                      if linea == 1:
                          P_Tipo1[NMovAct[linea-1]-1] = P_Tipo1[ordenM9_T1[NMovAct[linea-1]-1]-1]
                          P_Tipo2[NMovAct[linea-1]-1] = P_Tipo2[ordenM9_T2[NMovAct[linea-1]-1]-1]
                      end
                    else:
                      $ 709 "ElseIf Rec_Mosaico[Programa_1-1]≟10"
                      if (Rec_Mosaico[Programa_1-1] == 10):
                        $ 710 "Mosaico 10"
                        $ 716 "Script: mosaico10.script"
                        #MOSAICO 10
                        #P_Tipo1 y P_Tipo2 tienen que venir ya relativizados del asistente!

                        if ModificarMos == True:

                        	P_Tipo1_Mos10 = P_Tipo1
                        	P_Tipo2_Mos10 = P_Tipo2
                        	ordenM10_T1 = orden_T1
                        	ordenM10_T2 = orden_T2

                        end

                        ModificarMos = False

                        P_Tipo1 = P_Tipo1_Mos10
                        P_Tipo2 = P_Tipo2_Mos10


                        #En caso de que actualice movimientos de 2 en 2 (modificación de mosaico o crear nuevo)
                        if Cogida2en2 == True:

                        	Movs2en2_M10_T1 = Movs2en2_Tipo1
                        	Movs2en2_M10_T2 = Movs2en2_Tipo2

                        end

                        Cogida2en2 = False

                        #Siempre, si hay algún movimiento doble, actualizo si el movimiento actual lo es o no
                        if Rec_Cogida2en2[Programa-1] == True:
                        	if Rec_TipoCapa[NCapaAct[linea-1]-1] == 1:
                        		Movs2en2 = Movs2en2_M10_T1
                        		if linea == 1:
                        			Movs2en2[NMovAct[linea-1]-1] = Movs2en2[ordenM10_T1[NMovAct[linea-1]-1]-1]
                        		end
                        	else:
                        		Movs2en2 = Movs2en2_M10_T2
                        		if linea == 1:
                        			Movs2en2[NMovAct[linea-1]-1] = Movs2en2[ordenM10_T2[NMovAct[linea-1]-1]-1]
                        		end
                        	end
                        else:
                        	Movs2en2[NMovAct[linea-1]-1] = False
                        end

                        if linea == 1:
                            P_Tipo1[NMovAct[linea-1]-1] = P_Tipo1[ordenM10_T1[NMovAct[linea-1]-1]-1]
                            P_Tipo2[NMovAct[linea-1]-1] = P_Tipo2[ordenM10_T2[NMovAct[linea-1]-1]-1]
                        end
                      else:
                        $ 717 "ElseIf Rec_Mosaico[Programa_1-1]≟11"
                        if (Rec_Mosaico[Programa_1-1] == 11):
                          $ 718 "Mosaico 11"
                          $ 724 "Script: mosaico11.script"
                          #MOSAICO 10
                          #P_Tipo1 y P_Tipo2 tienen que venir ya relativizados del asistente!

                          if ModificarMos == True:

                          	P_Tipo1_Mos11 = P_Tipo1
                          	P_Tipo2_Mos11 = P_Tipo2
                          	ordenM11_T1 = orden_T1
                          	ordenM11_T2 = orden_T2

                          end

                          ModificarMos = False

                          P_Tipo1 = P_Tipo1_Mos11
                          P_Tipo2 = P_Tipo2_Mos11


                          #En caso de que actualice movimientos de 2 en 2 (modificación de mosaico o crear nuevo)
                          if Cogida2en2 == True:

                          	Movs2en2_M11_T1 = Movs2en2_Tipo1
                          	Movs2en2_M11_T2 = Movs2en2_Tipo2

                          end

                          Cogida2en2 = False

                          #Siempre, si hay algún movimiento doble, actualizo si el movimiento actual lo es o no
                          if Rec_Cogida2en2[Programa_1-1] == True:
                          	if Rec_TipoCapa[NCapaAct[linea-1]-1] == 1:
                          		Movs2en2 = Movs2en2_M11_T1
                          		if linea == 1:
                          			Movs2en2[NMovAct[linea-1]-1] = Movs2en2[ordenM11_T1[NMovAct[linea-1]-1]-1]
                          		end
                          	else:
                          		Movs2en2 = Movs2en2_M11_T2
                          		if linea == 1:
                          			Movs2en2[NMovAct[linea-1]-1] = Movs2en2[ordenM11_T2[NMovAct[linea-1]-1]-1]
                          		end
                          	end
                          else:
                          	Movs2en2[NMovAct[linea-1]-1] = False
                          end

                          if linea == 1:
                              P_Tipo1[NMovAct[linea-1]-1] = P_Tipo1[ordenM11_T1[NMovAct[linea-1]-1]-1]
                              P_Tipo2[NMovAct[linea-1]-1] = P_Tipo2[ordenM11_T2[NMovAct[linea-1]-1]-1]
                          end
                        else:
                          $ 725 "ElseIf Rec_Mosaico[Programa_1-1]≟12"
                          if (Rec_Mosaico[Programa_1-1] == 12):
                            $ 726 "Mosaico 12"
                            $ 796 "Script: mosaico12.script"
                            #MOSAICO 10
                            #P_Tipo1 y P_Tipo2 tienen que venir ya relativizados del asistente!

                            if ModificarMos == True:

                            	P_Tipo1_Mos12 = P_Tipo1
                            	P_Tipo2_Mos12 = P_Tipo2
                            	ordenM12_T1 = orden_T1
                            	ordenM12_T2 = orden_T2

                            end

                            ModificarMos = False

                            P_Tipo1 = P_Tipo1_Mos12
                            P_Tipo2 = P_Tipo2_Mos12


                            #En caso de que actualice movimientos de 2 en 2 (modificación de mosaico o crear nuevo)
                            if Cogida2en2 == True:

                            	Movs2en2_M12_T1 = Movs2en2_Tipo1
                            	Movs2en2_M12_T2 = Movs2en2_Tipo2

                            end

                            Cogida2en2 = False

                            #Siempre, si hay algún movimiento doble, actualizo si el movimiento actual lo es o no
                            if Rec_Cogida2en2[Programa_1-1] == True:
                            	if Rec_TipoCapa[NCapaAct[linea-1]-1] == 1:
                            		Movs2en2 = Movs2en2_M12_T1
                            		if linea == 1:
                            			Movs2en2[NMovAct[linea-1]-1] = Movs2en2[ordenM12_T1[NMovAct[linea-1]-1]-1]
                            		end
                            	else:
                            		Movs2en2 = Movs2en2_M12_T2
                            		if linea == 1:
                            			Movs2en2[NMovAct[linea-1]-1] = Movs2en2[ordenM12_T2[NMovAct[linea-1]-1]-1]
                            		end
                            	end
                            else:
                            	Movs2en2[NMovAct[linea-1]-1] = False
                            end

                            if linea == 1:
                                P_Tipo1[NMovAct[linea-1]-1] = P_Tipo1[ordenM12_T1[NMovAct[linea-1]-1]-1]
                                P_Tipo2[NMovAct[linea-1]-1] = P_Tipo2[ordenM12_T2[NMovAct[linea-1]-1]-1]
                            end
                          else:
                            $ 797 "Else" "noBreak"
                            $ 798 "Popup: Número de mosaico elegido no válido. Contacta con Geniotic."
                            popup("Número de mosaico elegido no válido. Contacta con Geniotic.", "Mensaje", False, False, blocking=True)
                            $ 799 "Halt"
                            halt
                          end
                        end
                      end
                    end
                  end
                end
              end
            end
          end
        end
      end
    end
  end
  def Cambios():
    $ 800 "Cambios" "noBreak"
    $ 801 "StepCode = 5"
    StepCode = 5
    $ 802 "If CambioPrograma"
    if (CambioPrograma):
      $ 803 "write_output_boolean_register(5,False)"
      write_output_boolean_register(5,False)
      $ 804 "'CambiosPrograma = False'"
      # 'CambiosPrograma = False'
      $ 809 "PonerCarton = [False,False]"
      PonerCarton = [False,False]
      $ 810 "Confirmacion = request_boolean_from_primary_client(' Al cambiar de programa se inicializan los contadores, ¿quieres continuar? ')"
      Confirmacion = request_boolean_from_primary_client(" Al cambiar de programa se inicializan los contadores, ¿quieres continuar? ")
      $ 811 "If Confirmacion"
      if (Confirmacion):
        $ 812 "Confirmacion = False"
        Confirmacion = False
        $ 813 "If (NCapaAct[0] ≠1 or NMovAct[0]≠1)"
        if ((NCapaAct[0]  != 1  or  NMovAct[0] != 1)):
          $ 814 "palet_completo(0)"
          palet_completo(0)
        end
        $ 815 "If (NCapaAct[1] ≠1 or NMovAct[1]≠1)"
        if ((NCapaAct[1]  != 1  or  NMovAct[1] != 1)):
          $ 816 "palet_completo(1)"
          palet_completo(1)
        end
        $ 817 "Wait: 0.01"
        sleep(0.01)
        $ 818 "aux = request_integer_from_primary_client('Elige programa [1-12]')"
        aux = request_integer_from_primary_client("Elige programa [1-12]")
        $ 819 "Wait: 0.01"
        sleep(0.01)
        $ 820 "Loop aux<1 or aux>12"
        while (aux<1 or aux>12):
          $ 821 "aux = request_integer_from_primary_client('Elige programa válido [1-12]')"
          aux = request_integer_from_primary_client("Elige programa válido [1-12]")
          $ 822 "sync()"
          sync()
        end
        $ 823 "If Rec_Mosaico[aux-1]≟0"
        if (Rec_Mosaico[aux-1] == 0):
          $ 824 "popup(' Programa vacío. Creálo o cambia a otro programa', title = ' Programa vacío', blocking = True)"
          popup(" Programa vacío. Creálo o cambia a otro programa", title = " Programa vacío", blocking = True)
        else:
          $ 825 "Else" "noBreak"
          $ 826 "Programa_1 = aux"
          Programa_1 = aux
        end
        $ 827 "NPaletAct = 0"
        NPaletAct = 0
        $ 828 "pop_up('¡Cambios finalizados!',3,False)"
        pop_up("¡Cambios finalizados!",3,False)
      end
    end
    $ 829 "If CambiosAvanzados"
    if (CambiosAvanzados):
      $ 830 "write_output_boolean_register(6,False)"
      write_output_boolean_register(6,False)
      $ 831 "'CambiosAvanzados = False'"
      # 'CambiosAvanzados = False'
      $ 832 "movej(Home_q,0.5,0.5,0,0)"
      movej(Home_q,0.5,0.5,0,0)
      $ 836 "aux = request_integer_from_primary_client(' Introduce la contraseña ')"
      aux = request_integer_from_primary_client(" Introduce la contraseña ")
      $ 837 "If aux≟1234"
      if (aux == 1234):
        $ 838 "Cambio_2≔0"
        global Cambio_2=0
        $ 839 "Loop Cambio_2≟0"
        while (Cambio_2 == 0):
          $ 840 "Cambio = request_integer_from_primary_client('Modificar programa [1], cambiar contadores [2] o ajustar un mov [3]?')"
          Cambio = request_integer_from_primary_client("Modificar programa [1], cambiar contadores [2] o ajustar un mov [3]?")
          $ 841 "Wait: 0.5"
          sleep(0.5)
          $ 842 "Loop Cambio<1 or Cambio>3"
          while (Cambio<1  or  Cambio>3):
            $ 843 "Cambio = request_integer_from_primary_client('Modificar programa [1], cambiar contadores [2] o ajustar un mov [3]?')"
            Cambio = request_integer_from_primary_client("Modificar programa [1], cambiar contadores [2] o ajustar un mov [3]?")
            $ 844 "sync()"
            sync()
          end
          $ 845 "If Cambio≟1"
          if (Cambio == 1):
            $ 846 "StepCode = 6"
            StepCode = 6
            $ 847 "Modificar_Programa"
            $ 848 "Confirmacion = request_boolean_from_primary_client(' Al cambiar de programa se inicializan los contadores, ¿quieres continuar? ')"
            Confirmacion = request_boolean_from_primary_client(" Al cambiar de programa se inicializan los contadores, ¿quieres continuar? ")
            $ 849 "If Confirmacion"
            if (Confirmacion):
              $ 850 "Confirmacion = False"
              Confirmacion = False
              $ 851 "If (NCapaAct[0] ≠1 or NMovAct[0]≠1)"
              if ((NCapaAct[0]  != 1  or  NMovAct[0] != 1)):
                $ 852 "palet_completo(0)"
                palet_completo(0)
              end
              $ 853 "If (NCapaAct[1] ≠1 or NMovAct[1]≠1)"
              if ((NCapaAct[1]  != 1  or  NMovAct[1] != 1)):
                $ 854 "palet_completo(1)"
                palet_completo(1)
              end
              $ 855 "Wait: 0.01"
              sleep(0.01)
              $ 856 "aux = request_integer_from_primary_client('Elige programa [1-12]')"
              aux = request_integer_from_primary_client("Elige programa [1-12]")
              $ 857 "Wait: 0.01"
              sleep(0.01)
              $ 858 "Loop aux<1 or aux>12"
              while (aux<1 or aux>12):
                $ 859 "aux = request_integer_from_primary_client('Elige programa válido [1-12]')"
                aux = request_integer_from_primary_client("Elige programa válido [1-12]")
                $ 860 "sync()"
                sync()
              end
              $ 861 "Loop Rec_Mosaico[aux-1]≟0 and ProgNuevo≟ False "
              while (Rec_Mosaico[aux-1] == 0  and  ProgNuevo ==   False  ):
                $ 862 "ProgNuevo = request_boolean_from_primary_client('Programa vacío. ¿Quieres crear uno nuevo [Sí] o elegir otro programa a modificar [No]?')"
                ProgNuevo = request_boolean_from_primary_client("Programa vacío. ¿Quieres crear uno nuevo [Sí] o elegir otro programa a modificar [No]?")
                $ 863 "If ProgNuevo≟ False "
                if (ProgNuevo ==   False  ):
                  $ 864 "aux = request_integer_from_primary_client('Elige programa [1-12]')"
                  aux = request_integer_from_primary_client("Elige programa [1-12]")
                  $ 865 "Loop aux<1 or aux>12"
                  while (aux<1 or aux>12):
                    $ 866 "aux = request_integer_from_primary_client('Elige programa válido [1-12]')"
                    aux = request_integer_from_primary_client("Elige programa válido [1-12]")
                    $ 867 "sync()"
                    sync()
                  end
                end
                $ 868 "sync()"
                sync()
              end
              $ 869 "ProgNuevo = False"
              ProgNuevo = False
              $ 870 "NPaletAct = 0"
              NPaletAct = 0
              $ 871 "Programa_1 = aux"
              Programa_1 = aux
              $ 872 "Modificaciones"
              $ 873 "aux_bool = request_boolean_from_primary_client(' ¿Quieres modificar el punto de cogida?')"
              aux_bool = request_boolean_from_primary_client(" ¿Quieres modificar el punto de cogida?")
              $ 874 "If aux_bool"
              if (aux_bool):
                $ 875 "freedrive_mode()"
                freedrive_mode()
                $ 876 "popup('Ve al punto y presiona Continuar', 'Punto cogida', False, False, blocking=True)"
                popup("Ve al punto y presiona Continuar", "Punto cogida", False, False, blocking=True)
                $ 877 "end_freedrive_mode()"
                end_freedrive_mode()
                $ 878 "PuntosCogida[Programa_1-1]=get_actual_tcp_pose()"
                PuntosCogida[Programa_1-1]= get_actual_tcp_pose ()
                $ 879 "popup('Mueve el robot a un sitio seguro antes de ir a Home', 'Mensaje', False, False, blocking=True)"
                popup("Mueve el robot a un sitio seguro antes de ir a Home", "Mensaje", False, False, blocking=True)
                $ 880 "movej(Home_q,0.5,0.5,0,0)"
                movej(Home_q,0.5,0.5,0,0)
              end
              $ 881 "aux=request_integer_from_primary_client('Largo producto (mm)')"
              aux=request_integer_from_primary_client("Largo producto (mm)")
              $ 882 "Rec_LargoPrd[Programa_1-1]=aux"
              Rec_LargoPrd[Programa_1-1]=aux
              $ 883 "Wait: 0.5"
              sleep(0.5)
              $ 884 "aux=request_integer_from_primary_client('Ancho producto (mm)')"
              aux=request_integer_from_primary_client("Ancho producto (mm)")
              $ 885 "Rec_AnchoPrd[Programa_1-1]=aux"
              Rec_AnchoPrd[Programa_1-1]=aux
              $ 886 "Wait: 0.5"
              sleep(0.5)
              $ 887 "aux_float=request_float_from_primary_client('Alto producto (mm)')"
              aux_float=request_float_from_primary_client("Alto producto (mm)")
              $ 888 "Rec_AltoPrd[Programa_1-1]=aux_float"
              Rec_AltoPrd[Programa_1-1]=aux_float
              $ 889 "Wait: 0.5"
              sleep(0.5)
              $ 890 "aux=request_integer_from_primary_client('Número de movimientos por capa')"
              aux=request_integer_from_primary_client("Número de movimientos por capa")
              $ 891 "Rec_NMovsCapa[Programa_1-1]=aux"
              Rec_NMovsCapa[Programa_1-1]=aux
              $ 892 "Wait: 0.5"
              sleep(0.5)
              $ 893 "aux=request_integer_from_primary_client('Número de capas totales')"
              aux=request_integer_from_primary_client("Número de capas totales")
              $ 894 "Rec_NCapasTot[Programa_1-1]=aux"
              Rec_NCapasTot[Programa_1-1]=aux
              $ 895 "Wait: 0.5"
              sleep(0.5)
              $ 896 "aux_bool=request_boolean_from_primary_client('¿Capas trabadas?')"
              aux_bool=request_boolean_from_primary_client("¿Capas trabadas?")
              $ 897 "Rec_CapasTrab[Programa_1-1]=aux_bool"
              Rec_CapasTrab[Programa_1-1]=aux_bool
              $ 898 "Wait: 0.5"
              sleep(0.5)
              $ 899 "aux_float=request_float_from_primary_client('Peso producto (kg)')"
              aux_float=request_float_from_primary_client("Peso producto (kg)")
              $ 900 "Rec_PesoPrd[Programa_1-1]=aux_float"
              Rec_PesoPrd[Programa_1-1]=aux_float
              $ 901 "Wait: 0.5"
              sleep(0.5)
              $ 902 "aux_bool=request_boolean_from_primary_client('¿Quieres usar un mosaico existente [Sí] o modificar/crear un mosaico [No]?')"
              aux_bool=request_boolean_from_primary_client("¿Quieres usar un mosaico existente [Sí] o modificar/crear un mosaico [No]?")
              $ 903 "ModificarMos = not(aux_bool)"
              ModificarMos = not(aux_bool)
              $ 904 "Wait: 0.5"
              sleep(0.5)
              $ 905 "aux=request_integer_from_primary_client('Elige un mosaico [1-12]')"
              aux=request_integer_from_primary_client("Elige un mosaico [1-12]")
              $ 906 "Loop aux<1 or aux>12"
              while (aux<1  or  aux>12):
                $ 907 "aux=request_integer_from_primary_client('Elige un mosaico válido [1-12]')"
                aux=request_integer_from_primary_client("Elige un mosaico válido [1-12]")
                $ 908 "sync()"
                sync()
              end
              $ 909 "Wait: 0.5"
              sleep(0.5)
              $ 910 "Rec_Mosaico[Programa_1-1]=aux"
              Rec_Mosaico[Programa_1-1]=aux
              $ 911 "Modificar mosaico"
              $ 912 "If ModificarMos"
              if (ModificarMos):
                $ 913 "i≔0"
                global i=0
                $ 914 "popup('Presiona Continuar para grabar los movimientos de la primera capa', 'Ajuste mosaico tipo capa 1', False, False, blocking=True)"
                popup("Presiona Continuar para grabar los movimientos de la primera capa", "Ajuste mosaico tipo capa 1", False, False, blocking=True)
                $ 915 "Loop i<Rec_NMovsCapa[Programa_1-1]"
                while (i<Rec_NMovsCapa[Programa_1-1]):
                  $ 916 "freedrive_mode()"
                  freedrive_mode()
                  $ 917 "popup('Mueve el robot al movimiento ' + to_str(i+1) + ' y presiona Continuar', title = ' Ajuste mosaico tipo capa 1', blocking = True)"
                  popup("Mueve el robot al movimiento " + to_str(i+1) + " y presiona Continuar", title = " Ajuste mosaico tipo capa 1", blocking = True)
                  $ 918 "end_freedrive_mode()"
                  end_freedrive_mode()
                  $ 919 "P_Tipo1[i] = get_actual_tcp_pose()"
                  P_Tipo1[i] =  get_actual_tcp_pose ()
                  $ 920 "i = i + 1"
                  i = i + 1
                  $ 921 "sync()"
                  sync()
                end
                $ 922 "i=0"
                i=0
                $ 923 "If Rec_CapasTrab[Programa_1-1]"
                if (Rec_CapasTrab[Programa_1-1]):
                  $ 924 "popup('Presiona Continuar para grabar los movimientos de la segunda capa', 'Ajuste mosaico tipo capa 2', False, False, blocking=True)"
                  popup("Presiona Continuar para grabar los movimientos de la segunda capa", "Ajuste mosaico tipo capa 2", False, False, blocking=True)
                  $ 925 "Loop i<Rec_NMovsCapa[Programa_1-1]"
                  while (i<Rec_NMovsCapa[Programa_1-1]):
                    $ 926 "freedrive_mode()"
                    freedrive_mode()
                    $ 927 "popup('Mueve el robot al movimiento ' + to_str(i+1) + ' y presiona Continuar', title = ' Ajuste mosaico tipo capa 2', blocking = True)"
                    popup("Mueve el robot al movimiento " + to_str(i+1) + " y presiona Continuar", title = " Ajuste mosaico tipo capa 2", blocking = True)
                    $ 928 "end_freedrive_mode()"
                    end_freedrive_mode()
                    $ 929 "P_Tipo2[i] = get_actual_tcp_pose()"
                    P_Tipo2[i] =  get_actual_tcp_pose ()
                    $ 930 "i = i + 1"
                    i = i + 1
                    $ 931 "sync()"
                    sync()
                  end
                end
                $ 932 "freedrive_mode()"
                freedrive_mode()
                $ 933 "popup('Mueve el robot a un sitio seguro antes de ir a Home', 'Mensaje', False, False, blocking=True)"
                popup("Mueve el robot a un sitio seguro antes de ir a Home", "Mensaje", False, False, blocking=True)
                $ 934 "end_freedrive_mode()"
                end_freedrive_mode()
                $ 935 "Wait: 0.5"
                sleep(0.5)
                $ 936 "Script: Relativizar.script"
                #Tras grabar los puntos
                local k = 0
                while k < 25:
                    P_Tipo1[k] = pose_trans(Pbf,P_Tipo1[k])
                    P_Tipo2[k] = pose_trans(Pbf,P_Tipo2[k])
                    k = k + 1
                end
                $ 937 "movej(Home_q,0.5,0.5,0,0)"
                movej(Home_q,0.5,0.5,0,0)
                $ 938 "Orden"
                $ 939 "aux = 0"
                aux = 0
                $ 940 "popup('Al presionar Continuar vamos a configurar los mosaicos de la línea 1', 'Mensaje', False, False, blocking=True)"
                popup("Al presionar Continuar vamos a configurar los mosaicos de la línea 1", "Mensaje", False, False, blocking=True)
                $ 941 "popup('Presiona Continuar para indicar el orden de los movimientos de la primera capa', 'Mensaje', False, False, blocking=True)"
                popup("Presiona Continuar para indicar el orden de los movimientos de la primera capa", "Mensaje", False, False, blocking=True)
                $ 942 "Loop aux<Rec_NMovsCapa[Programa_1-1]"
                while (aux<Rec_NMovsCapa[Programa_1-1]):
                  $ 943 "orden_T1[aux] = request_integer_from_primary_client(' El movimiento número ' + to_str(aux+1) + ' de la línea 1, ¿con qué número de movimiento se corresponde de la línea 2?')"
                  orden_T1[aux] = request_integer_from_primary_client(" El movimiento número " + to_str(aux+1) + " de la línea 1, ¿con qué número de movimiento se corresponde de la línea 2?")
                  $ 944 "aux = aux +1"
                  aux = aux +1
                  $ 945 "sync()"
                  sync()
                end
                $ 946 "If Rec_CapasTrab[Programa_1-1]"
                if (Rec_CapasTrab[Programa_1-1]):
                  $ 947 "popup('Presiona Continuar para indicar el orden de los movimientos de la segunda capa', 'Mensaje', False, False, blocking=True)"
                  popup("Presiona Continuar para indicar el orden de los movimientos de la segunda capa", "Mensaje", False, False, blocking=True)
                  $ 948 "aux = 0"
                  aux = 0
                  $ 949 "Loop aux<Rec_NMovsCapa[Programa_1-1]"
                  while (aux<Rec_NMovsCapa[Programa_1-1]):
                    $ 950 "orden_T2[aux] = request_integer_from_primary_client(' El movimiento número ' + to_str(aux+1) + ' de la línea 1, ¿con qué número de movimiento se corresponde de la línea 2?')"
                    orden_T2[aux] = request_integer_from_primary_client(" El movimiento número " + to_str(aux+1) + " de la línea 1, ¿con qué número de movimiento se corresponde de la línea 2?")
                    $ 951 "aux = aux +1"
                    aux = aux +1
                    $ 952 "sync()"
                    sync()
                  end
                end
                $ 953 "Cogida2en2=request_boolean_from_primary_client('¿Hay movimientos dobles?')"
                Cogida2en2=request_boolean_from_primary_client("¿Hay movimientos dobles?")
                $ 954 "Rec_Cogida2en2[Programa_1-1]=Cogida2en2"
                Rec_Cogida2en2[Programa_1-1]=Cogida2en2
                $ 955 "Wait: 0.5"
                sleep(0.5)
                $ 956 "Movimientos de 2 en 2"
                $ 957 "If Cogida2en2"
                if (Cogida2en2):
                  $ 958 "aux=request_integer_from_primary_client('¿Cuántos movimientos son dobles?')"
                  aux=request_integer_from_primary_client("¿Cuántos movimientos son dobles?")
                  $ 959 "Loop aux<1 or aux>Rec_NMovsCapa[Programa_1-1]"
                  while (aux<1  or  aux>Rec_NMovsCapa[Programa_1-1]):
                    $ 960 "aux=request_integer_from_primary_client('¿Cuántos movimientos son dobles?')"
                    aux=request_integer_from_primary_client("¿Cuántos movimientos son dobles?")
                    $ 961 "sync()"
                    sync()
                  end
                  $ 962 "aux_2=0"
                  aux_2=0
                  $ 963 "Loop aux_2<aux"
                  while (aux_2<aux):
                    $ 964 "aux_3=request_integer_from_primary_client('Indicar número del siguiente movimiento doble (primera capa)')"
                    aux_3=request_integer_from_primary_client("Indicar número del siguiente movimiento doble (primera capa)")
                    $ 965 "sync()"
                    sync()
                    $ 966 "Loop aux_3<1 or aux_3>Rec_NMovsCapa[Programa_1-1]"
                    while (aux_3<1  or  aux_3>Rec_NMovsCapa[Programa_1-1]):
                      $ 967 "aux_3=request_integer_from_primary_client('Número de movimiento doble incorrecto. Prueba otra vez:')"
                      aux_3=request_integer_from_primary_client("Número de movimiento doble incorrecto. Prueba otra vez:")
                      $ 968 "sync()"
                      sync()
                    end
                    $ 969 "Movs2en2_Tipo1[aux_3-1]= True "
                    Movs2en2_Tipo1[aux_3-1]=  True
                    $ 970 "aux_2=aux_2+1"
                    aux_2=aux_2+1
                  end
                  $ 971 "If Rec_CapasTrab[Programa_1-1]"
                  if (Rec_CapasTrab[Programa_1-1]):
                    $ 972 "aux_2=0"
                    aux_2=0
                    $ 973 "Loop aux_2<aux"
                    while (aux_2<aux):
                      $ 974 "aux_3=request_integer_from_primary_client('Indicar número del siguiente movimiento doble (segunda capa)')"
                      aux_3=request_integer_from_primary_client("Indicar número del siguiente movimiento doble (segunda capa)")
                      $ 975 "sync()"
                      sync()
                      $ 976 "Loop aux_3<1 or aux_3>Rec_NMovsCapa[Programa_1-1]"
                      while (aux_3<1  or  aux_3>Rec_NMovsCapa[Programa_1-1]):
                        $ 977 "aux_3=request_integer_from_primary_client('Número de movimiento doble incorrecto. Prueba otra vez:')"
                        aux_3=request_integer_from_primary_client("Número de movimiento doble incorrecto. Prueba otra vez:")
                        $ 978 "sync()"
                        sync()
                      end
                      $ 979 "Movs2en2_Tipo2[aux_3-1]= True "
                      Movs2en2_Tipo2[aux_3-1]=  True
                      $ 980 "aux_2=aux_2+1"
                      aux_2=aux_2+1
                    end
                  end
                else:
                  $ 981 "Else" "noBreak"
                  $ 982 "aux_bool=request_boolean_from_primary_client('¿Es necesario activar los 2 circuitos de vacío para coger este producto?')"
                  aux_bool=request_boolean_from_primary_client("¿Es necesario activar los 2 circuitos de vacío para coger este producto?")
                  $ 983 "Rec_2Vacios[Programa_1-1] = aux_bool"
                  Rec_2Vacios[Programa_1-1] = aux_bool
                end
              end
            end
          else:
            $ 984 "ElseIf Cambio≟2"
            if (Cambio == 2):
              $ 985 "StepCode = 7"
              StepCode = 7
              $ 986 "Cambio_Contadores"
              $ 987 "aux = request_integer_from_primary_client('Línea [1 - 2]')"
              aux = request_integer_from_primary_client("Línea [1 - 2]")
              $ 988 "Wait: 0.5"
              sleep(0.5)
              $ 989 "Loop aux<1 or aux>2"
              while (aux<1  or  aux>2):
                $ 990 "aux = request_integer_from_primary_client('Línea [1 - 2]')"
                aux = request_integer_from_primary_client("Línea [1 - 2]")
                $ 991 "sync()"
                sync()
              end
              $ 992 "PonerCarton[aux-1] = False"
              PonerCarton[aux-1] = False
              $ 993 "CartonBase[aux-1] = True"
              CartonBase[aux-1] = True
              $ 994 "aux_2 = request_integer_from_primary_client(' Número de capa [1 - ' + to_str(Rec_NCapasTot[Programa_1-1]) +  ']')"
              aux_2 = request_integer_from_primary_client(" Número de capa [1 - " + to_str(Rec_NCapasTot[Programa_1-1]) +  "]")
              $ 995 "Wait: 0.5"
              sleep(0.5)
              $ 996 "Loop aux_2<1 or aux_2>Rec_NCapasTot[Programa_1-1]"
              while (aux_2<1  or  aux_2>Rec_NCapasTot[Programa_1-1]):
                $ 997 "aux_2 = request_integer_from_primary_client(' Número de capa [1 - ' + to_str(Rec_NCapasTot[Programa_1-1]) +  ']')"
                aux_2 = request_integer_from_primary_client(" Número de capa [1 - " + to_str(Rec_NCapasTot[Programa_1-1]) +  "]")
                $ 998 "sync()"
                sync()
              end
              $ 999 "NCapaAct[aux-1] = aux_2"
              NCapaAct[aux-1] = aux_2
              $ 1000 "aux_2= request_integer_from_primary_client(' Número de movimiento [1 - ' + to_str(Rec_NMovsCapa[Programa_1-1]) +  ']')"
              aux_2= request_integer_from_primary_client(" Número de movimiento [1 - " + to_str(Rec_NMovsCapa[Programa_1-1]) +  "]")
              $ 1001 "Wait: 0.5"
              sleep(0.5)
              $ 1002 "Loop aux_2<1 or aux_2>Rec_NMovsCapa[Programa_1-1]"
              while (aux_2<1  or  aux_2>Rec_NMovsCapa[Programa_1-1]):
                $ 1003 "aux_2= request_integer_from_primary_client(' Número de movimiento [1 - ' + to_str(Rec_NMovsCapa[Programa_1-1]) +  ']')"
                aux_2= request_integer_from_primary_client(" Número de movimiento [1 - " + to_str(Rec_NMovsCapa[Programa_1-1]) +  "]")
                $ 1004 "sync()"
                sync()
              end
              $ 1005 "NMovAct[aux-1] = aux_2"
              NMovAct[aux-1] = aux_2
            else:
              $ 1006 "ElseIf Cambio≟3"
              if (Cambio == 3):
                $ 1007 "StepCode = 8"
                StepCode = 8
                $ 1008 "Ajuste de un movimiento"
                $ 1009 "aux_bool = request_boolean_from_primary_client('¿Quieres ajustar un movimiento de dejada [Sí] o cogida [No]?')"
                aux_bool = request_boolean_from_primary_client("¿Quieres ajustar un movimiento de dejada [Sí] o cogida [No]?")
                $ 1010 "Wait: 0.5"
                sleep(0.5)
                $ 1011 "If aux_bool"
                if (aux_bool):
                  $ 1012 "If Rec_CapasTrab[Programa_1-1]≟ True "
                  if (Rec_CapasTrab[Programa_1-1] ==   True  ):
                    $ 1013 "Ajuste_TipoCapa = request_integer_from_primary_client('Elige el tipo de capa a ajustar [1 - 2]')"
                    Ajuste_TipoCapa = request_integer_from_primary_client("Elige el tipo de capa a ajustar [1 - 2]")
                    $ 1014 "Wait: 0.5"
                    sleep(0.5)
                    $ 1015 "Loop Ajuste_TipoCapa<1 or Ajuste_TipoCapa>2"
                    while (Ajuste_TipoCapa<1  or  Ajuste_TipoCapa>2):
                      $ 1016 "Ajuste_TipoCapa = request_integer_from_primary_client('Elige el tipo de capa a ajustar [1 - 2]')"
                      Ajuste_TipoCapa = request_integer_from_primary_client("Elige el tipo de capa a ajustar [1 - 2]")
                      $ 1017 "sync()"
                      sync()
                    end
                  else:
                    $ 1018 "Else" "noBreak"
                    $ 1019 "Ajuste_TipoCapa = 1"
                    Ajuste_TipoCapa = 1
                  end
                  $ 1020 "Ajuste_NumMov = request_integer_from_primary_client(' ¿Qué movimiento quieres ajustar? [1-' +to_str(Rec_NMovsCapa[Programa_1-1])+']')"
                  Ajuste_NumMov = request_integer_from_primary_client(" ¿Qué movimiento quieres ajustar? [1-" +to_str(Rec_NMovsCapa[Programa_1-1])+"]")
                  $ 1021 "Wait: 0.5"
                  sleep(0.5)
                  $ 1022 "Loop Ajuste_NumMov<1 or Ajuste_NumMov>Rec_NMovsCapa[Programa_1-1]"
                  while (Ajuste_NumMov<1  or  Ajuste_NumMov>Rec_NMovsCapa[Programa_1-1]):
                    $ 1023 "Ajuste_NumMov = request_integer_from_primary_client(' ¿Qué movimiento quieres ajustar? [1-' +to_str(Rec_NMovsCapa[Programa_1-1])+']')"
                    Ajuste_NumMov = request_integer_from_primary_client(" ¿Qué movimiento quieres ajustar? [1-" +to_str(Rec_NMovsCapa[Programa_1-1])+"]")
                    $ 1024 "sync()"
                    sync()
                  end
                  $ 1025 "AjusteX_dejada = request_float_from_primary_client(' Ajuste en X (mm)')"
                  AjusteX_dejada = request_float_from_primary_client(" Ajuste en X (mm)")
                  $ 1026 "Wait: 0.5"
                  sleep(0.5)
                  $ 1027 "AjusteY_dejada = request_float_from_primary_client(' Ajuste en Y (mm)')"
                  AjusteY_dejada = request_float_from_primary_client(" Ajuste en Y (mm)")
                  $ 1028 "Wait: 0.5"
                  sleep(0.5)
                  $ 1030 "AjusteDejada = True"
                  AjusteDejada = True
                else:
                  $ 1031 "Else" "noBreak"
                  $ 1032 "AjusteX_cogida = request_float_from_primary_client(' Ajuste en X (mm)')"
                  AjusteX_cogida = request_float_from_primary_client(" Ajuste en X (mm)")
                  $ 1033 "Wait: 0.5"
                  sleep(0.5)
                  $ 1034 "AjusteY_cogida = request_float_from_primary_client(' Ajuste en Y (mm)')"
                  AjusteY_cogida = request_float_from_primary_client(" Ajuste en Y (mm)")
                  $ 1035 "Wait: 0.5"
                  sleep(0.5)
                  $ 1037 "AjusteCogida = True"
                  AjusteCogida = True
                end
                $ 1038 "Script: AjustesUsuario.script"
                #Ajuste de un punto

                #COGIDA
                if AjusteCogida == True:

                    local PuntoAModificar = PuntosCogida[Programa_1-1]

                    #Ajustes en función del plano referencia
                    PuntoAModificar = pose_trans(Pbf,PuntoAModificar)

                    PuntoAModificar[0] = PuntoAModificar[0] + AjusteX_cogida/1000
                    PuntoAModificar[1] = PuntoAModificar[1] + AjusteY_cogida/1000

                    #Anular rotaciones en X e Y y ajuste en RZ
                    local rpy = rotvec2rpy([PuntoAModificar[3],PuntoAModificar[4],PuntoAModificar[5]])
                    rpy[0]=3.142
                    rpy[1]=0
                    rpy[2] = rpy[2] + d2r(AjusteRZ_cogida)
                    local rotvec = rpy2rotvec(rpy)
                    PuntoAModificar[3] = rotvec[0]
                    PuntoAModificar[4] = rotvec[1]
                    PuntoAModificar[5] = rotvec[2]

                    #Volver a coordenadas de la base (porque en cogida no tenemos base)
                    PuntoAModificar = pose_trans(wObjDejadaRef,PuntoAModificar)

                    PuntosCogida[Programa_1-1] = PuntoAModificar

                    AjusteCogida = False
                end

                #DEJADA
                if AjusteDejada == True:

                	if Rec_Mosaico[Programa_1-1] == 1:

                    		if Ajuste_TipoCapa == 1:
                        			local PuntoAModificar = P_Tipo1_Mos1[Ajuste_NumMov-1]
                    		elif Ajuste_TipoCapa == 2:
                        			local PuntoAModificar = P_Tipo2_Mos1[Ajuste_NumMov-1]
                    		end

                	elif Rec_Mosaico[Programa_1-1] == 2:

                    		if Ajuste_TipoCapa == 1:
                        			local PuntoAModificar = P_Tipo1_Mos2[Ajuste_NumMov-1]
                    		elif Ajuste_TipoCapa == 2:
                        			local PuntoAModificar = P_Tipo2_Mos2[Ajuste_NumMov-1]
                    		end

                	elif Rec_Mosaico[Programa_1-1] == 3:

                    		if Ajuste_TipoCapa == 1:
                        			local PuntoAModificar = P_Tipo1_Mos3[Ajuste_NumMov-1]
                    		elif Ajuste_TipoCapa == 2:
                        			local PuntoAModificar = P_Tipo2_Mos3[Ajuste_NumMov-1]
                    		end


                	elif Rec_Mosaico[Programa_1-1] == 4:

                    		if Ajuste_TipoCapa == 1:
                        			local PuntoAModificar = P_Tipo1_Mos4[Ajuste_NumMov-1]
                    		elif Ajuste_TipoCapa == 2:
                        			local PuntoAModificar = P_Tipo2_Mos4[Ajuste_NumMov-1]
                    		end

                	elif Rec_Mosaico[Programa_1-1] == 5:

                    		if Ajuste_TipoCapa == 1:
                        			local PuntoAModificar = P_Tipo1_Mos5[Ajuste_NumMov-1]
                    		elif Ajuste_TipoCapa == 2:
                        			local PuntoAModificar = P_Tipo2_Mos5[Ajuste_NumMov-1]
                    		end

                	elif Rec_Mosaico[Programa_1-1] == 6:

                    		if Ajuste_TipoCapa == 1:
                        			local PuntoAModificar = P_Tipo1_Mos6[Ajuste_NumMov-1]
                    		elif Ajuste_TipoCapa == 2:
                        			local PuntoAModificar = P_Tipo2_Mos6[Ajuste_NumMov-1]
                    		end

                	elif Rec_Mosaico[Programa_1-1] == 7:

                    		if Ajuste_TipoCapa == 1:
                        			local PuntoAModificar = P_Tipo1_Mos7[Ajuste_NumMov-1]
                    		elif Ajuste_TipoCapa == 2:
                        			local PuntoAModificar = P_Tipo2_Mos7[Ajuste_NumMov-1]
                    		end

                	elif Rec_Mosaico[Programa_1-1] == 8:

                    		if Ajuste_TipoCapa == 1:
                        			local PuntoAModificar = P_Tipo1_Mos8[Ajuste_NumMov-1]
                    		elif Ajuste_TipoCapa == 2:
                        			local PuntoAModificar = P_Tipo2_Mos8[Ajuste_NumMov-1]
                    		end

                	elif Rec_Mosaico[Programa_1-1] == 9:

                    		if Ajuste_TipoCapa == 1:
                        			local PuntoAModificar = P_Tipo1_Mos9[Ajuste_NumMov-1]
                    		elif Ajuste_TipoCapa == 2:
                        			local PuntoAModificar = P_Tipo2_Mos9[Ajuste_NumMov-1]
                    		end

                	elif Rec_Mosaico[Programa_1-1] == 10:

                    		if Ajuste_TipoCapa == 1:
                        			local PuntoAModificar = P_Tipo1_Mos10[Ajuste_NumMov-1]
                    		elif Ajuste_TipoCapa == 2:
                        			local PuntoAModificar = P_Tipo2_Mos10[Ajuste_NumMov-1]
                    		end

                               end

                    PuntoAModificar[0] = PuntoAModificar[0] + AjusteX_dejada/1000
                    PuntoAModificar[1] = PuntoAModificar[1] + AjusteY_dejada/1000

                    #Anular rotaciones en X e Y y ajuste en RZ
                    local rpy = rotvec2rpy([PuntoAModificar[3],PuntoAModificar[4],PuntoAModificar[5]])
                    rpy[0]=3.142
                    rpy[1]=0
                    rpy[2] = rpy[2] + d2r(AjusteRZ_dejada)
                    local rotvec = rpy2rotvec(rpy)
                    PuntoAModificar[3] = rotvec[0]
                    PuntoAModificar[4] = rotvec[1]
                    PuntoAModificar[5] = rotvec[2]


                	if Rec_Mosaico[Programa_1-1] == 1:

                    		if Ajuste_TipoCapa == 1:
                        			P_Tipo1_Mos1[Ajuste_NumMov-1] = PuntoAModificar
                    		elif Ajuste_TipoCapa == 2:
                        			P_Tipo2_Mos1[Ajuste_NumMov-1] = PuntoAModificar
                    		end

                	elif Rec_Mosaico[Programa_1-1] == 2:

                    		if Ajuste_TipoCapa == 1:
                        			P_Tipo1_Mos2[Ajuste_NumMov-1] = PuntoAModificar
                    		elif Ajuste_TipoCapa == 2:
                        			P_Tipo2_Mos2[Ajuste_NumMov-1] = PuntoAModificar
                    		end

                	elif Rec_Mosaico[Programa_1-1] == 3:

                    		if Ajuste_TipoCapa == 1:
                        			P_Tipo1_Mos3[Ajuste_NumMov-1] = PuntoAModificar
                    		elif Ajuste_TipoCapa == 2:
                        			P_Tipo2_Mos3[Ajuste_NumMov-1] = PuntoAModificar
                    		end


                	elif Rec_Mosaico[Programa_1-1] == 4:

                    		if Ajuste_TipoCapa == 1:
                        			P_Tipo1_Mos4[Ajuste_NumMov-1] = PuntoAModificar
                    		elif Ajuste_TipoCapa == 2:
                        			P_Tipo2_Mos4[Ajuste_NumMov-1] = PuntoAModificar
                    		end

                	elif Rec_Mosaico[Programa_1-1] == 5:

                    		if Ajuste_TipoCapa == 1:
                        			P_Tipo1_Mos5[Ajuste_NumMov-1] = PuntoAModificar
                    		elif Ajuste_TipoCapa == 2:
                        			P_Tipo2_Mos5[Ajuste_NumMov-1] = PuntoAModificar
                    		end


                	elif Rec_Mosaico[Programa_1-1] == 6:

                		if Ajuste_TipoCapa == 1:
                				P_Tipo1_Mos6[Ajuste_NumMov-1] = PuntoAModificar
                		elif Ajuste_TipoCapa == 2:
                				P_Tipo2_Mos6[Ajuste_NumMov-1] = PuntoAModificar
                		end


                	elif Rec_Mosaico[Programa_1-1] == 7:

                    		if Ajuste_TipoCapa == 1:
                        			P_Tipo1_Mos7[Ajuste_NumMov-1] = PuntoAModificar
                    		elif Ajuste_TipoCapa == 2:
                        			P_Tipo2_Mos7[Ajuste_NumMov-1] = PuntoAModificar
                    		end


                	elif Rec_Mosaico[Programa_1-1] == 8:

                		if Ajuste_TipoCapa == 1:
                				P_Tipo1_Mos8[Ajuste_NumMov-1] = PuntoAModificar
                		elif Ajuste_TipoCapa == 2:
                				P_Tipo2_Mos8[Ajuste_NumMov-1] = PuntoAModificar
                		end


                	elif Rec_Mosaico[Programa_1-1] == 9:

                		if Ajuste_TipoCapa == 1:
                				P_Tipo1_Mos9[Ajuste_NumMov-1] = PuntoAModificar
                		elif Ajuste_TipoCapa == 2:
                				P_Tipo2_Mos9[Ajuste_NumMov-1] = PuntoAModificar
                		end


                	elif Rec_Mosaico[Programa_1-1] == 10:

                		if Ajuste_TipoCapa == 1:
                				P_Tipo1_Mos10[Ajuste_NumMov-1] = PuntoAModificar
                		elif Ajuste_TipoCapa == 2:
                				P_Tipo2_Mos10[Ajuste_NumMov-1] = PuntoAModificar
                		end

                	end

                    AjusteDejada = False

                end
              end
            end
          end
          $ 1039 "Cambio_2 = request_integer_from_primary_client(' Realizar otra operacion: SI [0], NO [1]?')"
          Cambio_2 = request_integer_from_primary_client(" Realizar otra operacion: SI [0], NO [1]?")
          $ 1040 "Wait: 0.5"
          sleep(0.5)
        end
        $ 1041 "pop_up('¡Cambios finalizados!',3,False)"
        pop_up("¡Cambios finalizados!",3,False)
      else:
        $ 1042 "Else" "noBreak"
        $ 1043 "pop_up('Contraseña no válida',2,False)"
        pop_up("Contraseña no válida",2,False)
      end
    end
    $ 1044 "Script: Calculos_previos.script"
    global PCogida = PuntosCogida[Programa-1]
    global OffsetZPreCogida = 50
    global PPreCogida = PCogida
    global zPCogida = (AltoTransporte - AltoBaseRobot)/1000 + Rec_AltoPrd[Programa-1]/1000 - 3/1000 - 13/1000
    global zPPreCogida = zPCogida + OffsetZPreCogida/1000
    PPreCogida[2] = zPPreCogida
    #PPreCogida[2] = zPPreCogida - pos_bajada[linea-1]/1000
    $ 1045 "MoveJTrans(PPreCogida,Base_const,0.5,0.5,0,0)"
    MoveJTrans(PPreCogida,p[0.0,0.0,0.0,0.0,0.0,0.0],0.5,0.5,0,0)
  end
  $ 1 "BeforeStart"
  $ 2 "Script: ConfigRobot.script"
  ##########################CONFIGURACIÓN DE INICIO DEL ROBOT############################

  ##Aqui se configuran las partes del robot para deshabilitar o habilitar partes que no se vallan a utilizar. ##

  ##Para configurar el robot habilitaremos (True) o deshabilitaremos (false) la siguiente array en la parte indicada para ese componente o parte del programa##

  global ConfigRbt = [False,False,False,False,False,False,False,False,False,False,False,False,False,False,False,False]

  #####DESCRIPCIÓN DE ARRAY ConfigRbt[i]#####

  #ConfigRbt[1] -> habilitamos y deshabilitamos la columna del Robot#








  #NOTA: se puede añadir tantos elementos a la array como vallamos necesitando#
  $ 3 "Script: InitVariables.script"
  global retraso = 0.1
  global relleno = p[100,100,100,0,0,0]
  global PesoTool = 1.10
  global cog = [0,0,0]
  global cog_vacio = [0/1000,0/1000,0/1000]


  #Variables de trabajo
  global P_Tipo1 = [relleno,relleno,relleno,relleno,relleno,relleno,relleno,relleno,relleno,relleno,relleno,relleno,relleno,relleno,relleno,relleno,relleno,relleno,relleno,relleno,relleno,relleno,relleno,relleno,relleno,relleno,relleno,relleno,relleno,relleno,relleno,relleno,relleno,relleno,relleno,relleno,relleno,relleno,relleno,relleno]
  global P_Tipo2 = [relleno,relleno,relleno,relleno,relleno,relleno,relleno,relleno,relleno,relleno,relleno,relleno,relleno,relleno,relleno,relleno,relleno,relleno,relleno,relleno,relleno,relleno,relleno,relleno,relleno,relleno,relleno,relleno,relleno,relleno,relleno,relleno,relleno,relleno,relleno,relleno,relleno,relleno,relleno,relleno]

  global Movs2en2_Tipo1 = [False, False, False, False, False, False, False, False, False, False, False, False, False, False, False, False, False, False, False, False, False, False, False, False, False, False, False, False, False, False, False, False, False, False, False, False, False, False, False, False]
  global Movs2en2_Tipo2 = [False, False, False, False, False, False, False, False, False, False, False, False, False, False, False, False, False, False, False, False, False, False, False, False, False, False, False, False, False, False, False, False, False, False, False, False, False, False, False, False]
  global Movs2en2 = [False, False, False, False, False, False, False, False, False, False, False, False, False, False, False, False, False, False, False, False, False, False, False, False, False, False, False, False, False, False, False, False, False, False, False, False, False, False, False, False]

  global orden_T1 = [1, 1, 1, 1, 1, 1, 1, 1, 1, 1, 1, 1, 1, 1, 1, 1, 1, 1, 1, 1, 1, 1, 1, 1, 1, 1, 1, 1, 1, 1, 1, 1, 1, 1, 1, 1, 1, 1, 1, 1]
  global orden_T2 = [1, 1, 1, 1, 1, 1, 1, 1, 1, 1, 1, 1, 1, 1, 1, 1, 1, 1, 1, 1, 1, 1, 1, 1, 1, 1, 1, 1, 1, 1, 1, 1, 1, 1, 1, 1, 1, 1, 1, 1]

  #Variables de E/S
  global iFT1 = False
  global iFT2 = False
  global iAVISO_SAI = False		#Cambio RGR 24/11/2022,Nueva variabla para FiltroES#
  global iFT4 = False
  global iFT5 = False
  global iQM1 = False
  global iVF1 = False
  global iQM2 = False
  global iVF2 = False
  global iVAC1 = False
  global iVAC2 = False

  #oEV1 y oEV2 y oEV4 son de instalación para mantener el estado (por si se aborta el Programa_1)
  global oB1V = False
  global oB1R = False
  global oB2V = False
  global oB2R = False
  global oEV5 = False
  global oM1 = False
  global oM2 = False
  global oRP_ME = True

  global oVELM1 = 0.4
  global oVELM2 = 0.5

  #Temporizadores a la conexión y desconexión entradas
  global tON_FT1 = 5
  global tON_FT2 = 5
  global tON_AVISO_SAI = 2		#Cambio RGR 24/11/2022,Nueva variabla para FiltroES#
  global tON_FT4 = 2
  global tON_FT5 = 2
  global tON_QM1 = 0.5
  global tON_VF1 = 0.5
  global tON_QM2 = 0.5
  global tON_VF2 = 0.5


  global tOFF_FT1 = 0.5
  global tOFF_FT2 = 0.5
  global tOFF_AVISO_SAI = 0.5 		#Cambio RGR 24/11/2022,Nueva variabla para FiltroES#
  global tOFF_FT4 = 0.5
  global tOFF_FT5 = 0.5
  global tOFF_QM1 = 0.5
  global tOFF_VF1 = 0.5
  global tOFF_QM2 = 0.5
  global tOFF_VF2 = 0.5

  #Variables de transiciones de las secuencias

  #Variables de aviso
  global AvisoPaletCompletoL1 = False
  global AvisoPaletCompletoL2 = False
  global AvisoPaletL1 = False
  global AvisoPaletL2 = False
  global AvisoL1Deshab = False
  global AvisoL2Deshab = False
  global Aviso = False


  #Variables auxiliares
  global actual = p[0,0,0,0,0,0]
  global aux = 0
  global aux_2 = 0
  global aux_3 = 0
  global aux_bool = False
  global aux_float = 0.0
  global aux_string = ""

  #Variables asistente cambio de Programa_1
  global CambioPrograma = False
  global CambiosAvanzados = False
  global Confirmacion = False
  global ModificarMos = False
  global Cogida2en2 = False
  global ProgNuevo = False

  #Variables asistente ajuste de un movimiento
  global AjusteDejada = False
  global AjusteCogida =False
  global AjusteX_cogida = 0.0
  global AjusteY_cogida= 0.0
  global AjusteRZ_cogida = 0.0
  global AjusteX_dejada = 0.0
  global AjusteY_dejada= 0.0
  global AjusteRZ_dejada = 0.0
  global Ajuste_TipoCapa = 0
  global Ajuste_NumMov = 0

  #Variables columna
  global trigger_subida = False
  global trigger_bajada = False
  global trigger_0 = False

  #Resto variables
  global DescargarPal = [False, False]
  global ResetSec = False
  global PermisoBotones = False
  global StepCode = 0
  global off = 2 		#offset de la columna
  global Offset = 45 	#offset de aproximación
  global linea_ant = linea
  global Per_LineaDeshab = False

  global yPPerchDejada_min_array = [0,0]
  global yPPerchDejada_max_array = [0,0]
  global xPPerchDejada_array = [0,0]

  global Pbf = pose_inv(wObjDejadaRef)

  if reset_puntos == True:


  	P_Tipo1_Mos1 = [WP1_Mos1_T1_p,WP2_Mos1_T1_p,WP3_Mos1_T1_p,WP4_Mos1_T1_p,WP5_Mos1_T1_p,WP6_Mos1_T1_p,WP7_Mos1_T1_p,WP8_Mos1_T1_p,WP9_Mos1_T1_p,WP10_Mos1_T1_p,WP11_Mos1_T1_p,WP12_Mos1_T1_p,WP13_Mos1_T1_p,WP14_Mos1_T1_p,WP15_Mos1_T1_p,WP16_Mos1_T1_p,WP17_Mos1_T1_p,WP18_Mos1_T1_p,WP19_Mos1_T1_p,WP20_Mos1_T1_p,WP21_Mos1_T1_p,WP22_Mos1_T1_p,WP23_Mos1_T1_p,WP24_Mos1_T1_p,WP25_Mos1_T1_p,WP26_Mos1_T1_p,WP27_Mos1_T1_p,WP28_Mos1_T1_p,WP29_Mos1_T1_p,WP30_Mos1_T1_p,WP31_Mos1_T1_p,WP32_Mos1_T1_p,relleno,relleno,relleno,relleno,relleno,relleno,relleno,relleno]
  	P_Tipo2_Mos1 = [WP1_Mos1_T2_p,WP2_Mos1_T2_p,WP3_Mos1_T2_p,WP4_Mos1_T2_p,WP5_Mos1_T2_p,WP6_Mos1_T2_p,WP7_Mos1_T2_p,WP8_Mos1_T2_p,WP9_Mos1_T2_p,WP10_Mos1_T2_p,WP11_Mos1_T2_p,WP12_Mos1_T2_p,WP13_Mos1_T2_p,WP14_Mos1_T2_p,WP15_Mos1_T2_p,WP16_Mos1_T2_p,WP17_Mos1_T2_p,WP18_Mos1_T2_p,WP19_Mos1_T2_p,WP20_Mos1_T2_p,WP21_Mos1_T2_p,WP22_Mos1_T2_p,WP23_Mos1_T2_p,WP24_Mos1_T2_p,WP25_Mos1_T2_p,WP26_Mos1_T2_p,WP27_Mos1_T2_p,WP28_Mos1_T2_p,WP29_Mos1_T2_p,WP30_Mos1_T2_p,WP31_Mos1_T2_p,WP32_Mos1_T2_p,relleno,relleno,relleno,relleno,relleno,relleno,relleno,relleno]

  	#P_Tipo1_Mos1 = [WP1_Mos1_T1_p,WP2_Mos1_T1_p,WP3_Mos1_T1_p,WP4_Mos1_T1_p,WP5_Mos1_T1_p,WP6_Mos1_T1_p,WP7_Mos1_T1_p,WP8_Mos1_T1_p,relleno,relleno,relleno,relleno,relleno,relleno,relleno,relleno,relleno,relleno,relleno,relleno,relleno,relleno,relleno,relleno,relleno,relleno,relleno,relleno,relleno,relleno,relleno,relleno,relleno,relleno,relleno,relleno,relleno,relleno,relleno,relleno]
  	#P_Tipo2_Mos1 = [WP1_Mos1_T2_p,WP2_Mos1_T2_p,WP3_Mos1_T2_p,WP4_Mos1_T2_p,WP5_Mos1_T2_p,WP6_Mos1_T2_p,WP7_Mos1_T2_p,WP8_Mos1_T2_p,relleno,relleno,relleno,relleno,relleno,relleno,relleno,relleno,relleno,relleno,relleno,relleno,relleno,relleno,relleno,relleno,relleno,relleno,relleno,relleno,relleno,relleno,relleno,relleno,relleno,relleno,relleno,relleno,relleno,relleno,relleno,relleno

  	#P_Tipo1_Mos2 = [WP1_Mos2_T1_p,WP2_Mos2_T1_p,WP3_Mos2_T1_p,WP4_Mos2_T1_p,WP5_Mos2_T1_p,WP6_Mos2_T1_p,WP7_Mos2_T1_p,WP8_Mos2_T1_p,WP9_Mos2_T1_p,WP10_Mos2_T1_p,WP11_Mos2_T1_p,WP12_Mos2_T1_p,WP13_Mos2_T1_p,WP14_Mos2_T1_p,relleno,relleno,relleno,relleno,relleno,relleno,relleno,relleno,relleno,relleno,relleno,relleno,relleno,relleno,relleno,relleno,relleno,relleno,relleno,relleno,relleno,relleno,relleno,relleno,relleno,relleno]
  	#P_Tipo2_Mos2 = [WP1_Mos2_T2_p,WP2_Mos2_T2_p,WP3_Mos2_T2_p,WP4_Mos2_T2_p,WP5_Mos2_T2_p,WP6_Mos2_T2_p,WP7_Mos2_T2_p,WP8_Mos2_T2_p,WP9_Mos2_T2_p,WP10_Mos2_T2_p,WP11_Mos2_T2_p,WP12_Mos2_T2_p,WP13_Mos2_T2_p,WP14_Mos2_T2_p,relleno,relleno,relleno,relleno,relleno,relleno,relleno,relleno,relleno,relleno,relleno,relleno,relleno,relleno,relleno,relleno,relleno,relleno,relleno,relleno,relleno,relleno,relleno,relleno,relleno,relleno]

  	#P_Tipo1_Mos3 = [WP1_Mos3_T1_p,WP2_Mos3_T1_p,WP3_Mos3_T1_p,WP4_Mos3_T1_p,WP5_Mos3_T1_p,WP6_Mos3_T1_p,WP7_Mos3_T1_p,WP8_Mos3_T1_p,WP9_Mos3_T1_p,WP10_Mos3_T1_p,WP11_Mos3_T1_p,WP12_Mos3_T1_p,WP13_Mos3_T1_p,WP14_Mos3_T1_p,WP15_Mos3_T1_p,WP16_Mos3_T1_p,WP17_Mos3_T1_p,WP18_Mos3_T1_p,WP19_Mos3_T1_p,WP20_Mos3_T1_p,relleno,relleno,relleno,relleno,relleno,relleno,relleno,relleno,relleno,relleno,relleno,relleno,relleno,relleno,relleno,relleno,relleno,relleno,relleno,relleno]
  	#P_Tipo2_Mos3 = [WP1_Mos3_T2_p,WP2_Mos3_T2_p,WP3_Mos3_T2_p,WP4_Mos3_T2_p,WP5_Mos3_T2_p,WP6_Mos3_T2_p,WP7_Mos3_T2_p,WP8_Mos3_T2_p,WP9_Mos3_T2_p,WP10_Mos3_T2_p,WP11_Mos3_T2_p,WP12_Mos3_T2_p,WP13_Mos3_T2_p,WP14_Mos3_T2_p,WP15_Mos3_T2_p,WP16_Mos3_T2_p,WP17_Mos3_T2_p,WP18_Mos3_T2_p,WP19_Mos3_T2_p,WP20_Mos3_T2_p,relleno,relleno,relleno,relleno,relleno,relleno,relleno,relleno,relleno,relleno,relleno,relleno,relleno,relleno,relleno,relleno,relleno,relleno,relleno,relleno]

  	#P_Tipo1_Mos4 = [WP1_Mos4_T1_p,WP2_Mos4_T1_p,WP3_Mos4_T1_p,WP4_Mos4_T1_p,WP5_Mos4_T1_p,WP6_Mos4_T1_p,WP7_Mos4_T1_p,WP8_Mos4_T1_p,WP9_Mos4_T1_p,WP10_Mos4_T1_p,relleno,relleno,relleno,relleno,relleno,relleno,relleno,relleno,relleno,relleno,relleno,relleno,relleno,relleno,relleno,relleno,relleno,relleno,relleno,relleno,relleno,relleno,relleno,relleno,relleno,relleno,relleno,relleno,relleno,relleno]
  	#P_Tipo2_Mos4 = [WP1_Mos4_T2_p,WP2_Mos4_T2_p,WP3_Mos4_T2_p,WP4_Mos4_T2_p,WP5_Mos4_T2_p,WP6_Mos4_T2_p,WP7_Mos4_T2_p,WP8_Mos4_T2_p,WP9_Mos4_T2_p,WP10_Mos4_T2_p,relleno,relleno,relleno,relleno,relleno,relleno,relleno,relleno,relleno,relleno,relleno,relleno,relleno,relleno,relleno,relleno,relleno,relleno,relleno,relleno,relleno,relleno,relleno,relleno,relleno,relleno,relleno,relleno,relleno,relleno]

  	#P_Tipo1_Mos5 = [WP1_Mos5_T1_p,WP2_Mos5_T1_p,WP3_Mos5_T1_p,WP4_Mos5_T1_p,WP5_Mos5_T1_p,WP6_Mos5_T1_p,WP7_Mos5_T1_p,WP8_Mos5_T1_p,WP9_Mos5_T1_p,WP10_Mos5_T1_p,relleno,relleno,relleno,relleno,relleno,relleno,relleno,relleno,relleno,relleno,relleno,relleno,relleno,relleno,relleno,relleno,relleno,relleno,relleno,relleno,relleno,relleno,relleno,relleno,relleno,relleno,relleno,relleno,relleno,relleno]
  	#P_Tipo2_Mos5 = [WP1_Mos5_T2_p,WP2_Mos5_T2_p,WP3_Mos5_T2_p,WP4_Mos5_T2_p,WP5_Mos5_T2_p,WP6_Mos5_T2_p,WP7_Mos5_T2_p,WP8_Mos5_T2_p,WP9_Mos5_T2_p,WP10_Mos5_T2_p,relleno,relleno,relleno,relleno,relleno,relleno,relleno,relleno,relleno,relleno,relleno,relleno,relleno,relleno,relleno,relleno,relleno,relleno,relleno,relleno,relleno,relleno,relleno,relleno,relleno,relleno,relleno,relleno,relleno,relleno]

  	#P_Tipo1_Mos6 = [WP1_Mos6_T1_p,WP2_Mos6_T1_p,WP3_Mos6_T1_p,WP4_Mos6_T1_p,WP5_Mos6_T1_p,WP6_Mos6_T1_p,WP7_Mos6_T1_p,WP8_Mos6_T1_p,WP9_Mos6_T1_p,WP10_Mos6_T1_p,relleno,relleno,relleno,relleno,relleno,relleno,relleno,relleno,relleno,relleno,relleno,relleno,relleno,relleno,relleno,relleno,relleno,relleno,relleno,relleno,relleno,relleno,relleno,relleno,relleno,relleno,relleno,relleno,relleno,relleno]
  	#P_Tipo2_Mos6 = [WP1_Mos6_T2_p,WP2_Mos6_T2_p,WP3_Mos6_T2_p,WP4_Mos6_T2_p,WP5_Mos6_T2_p,WP6_Mos6_T2_p,WP7_Mos6_T2_p,WP8_Mos6_T2_p,WP9_Mos6_T2_p,WP10_Mos6_T2_p,relleno,relleno,relleno,relleno,relleno,relleno,relleno,relleno,relleno,relleno,relleno,relleno,relleno,relleno,relleno,relleno,relleno,relleno,relleno,relleno,relleno,relleno,relleno,relleno,relleno,relleno,relleno,relleno,relleno,relleno]

  	#P_Tipo1_Mos7 = [WP1_Mos7_T1_p,WP2_Mos7_T1_p,WP3_Mos7_T1_p,WP4_Mos7_T1_p,WP5_Mos7_T1_p,WP6_Mos7_T1_p,WP7_Mos7_T1_p,WP8_Mos7_T1_p,WP9_Mos7_T1_p,WP10_Mos7_T1_p,relleno,relleno,relleno,relleno,relleno,relleno,relleno,relleno,relleno,relleno,relleno,relleno,relleno,relleno,relleno,relleno,relleno,relleno,relleno,relleno,relleno,relleno,relleno,relleno,relleno,relleno,relleno,relleno,relleno,relleno]
  	#P_Tipo2_Mos7 = [WP1_Mos7_T2_p,WP2_Mos7_T2_p,WP3_Mos7_T2_p,WP4_Mos7_T2_p,WP5_Mos7_T2_p,WP6_Mos7_T2_p,WP7_Mos7_T2_p,WP8_Mos7_T2_p,WP9_Mos7_T2_p,WP10_Mos7_T2_p,relleno,relleno,relleno,relleno,relleno,relleno,relleno,relleno,relleno,relleno,relleno,relleno,relleno,relleno,relleno,relleno,relleno,relleno,relleno,relleno,relleno,relleno,relleno,relleno,relleno,relleno,relleno,relleno,relleno,relleno]

  	#P_Tipo1_Mos8 = [WP1_Mos8_T1_p,WP2_Mos8_T1_p,WP3_Mos8_T1_p,WP4_Mos8_T1_p,WP5_Mos8_T1_p,WP6_Mos8_T1_p,WP7_Mos8_T1_p,WP8_Mos8_T1_p,WP9_Mos8_T1_p,WP10_Mos8_T1_p,relleno,relleno,relleno,relleno,relleno,relleno,relleno,relleno,relleno,relleno,relleno,relleno,relleno,relleno,relleno,relleno,relleno,relleno,relleno,relleno,relleno,relleno,relleno,relleno,relleno,relleno,relleno,relleno,relleno,relleno]
  	#P_Tipo2_Mos8 = [WP1_Mos8_T2_p,WP2_Mos8_T2_p,WP3_Mos8_T2_p,WP4_Mos8_T2_p,WP5_Mos8_T2_p,WP6_Mos8_T2_p,WP7_Mos8_T2_p,WP8_Mos8_T2_p,WP9_Mos8_T2_p,WP10_Mos8_T2_p,relleno,relleno,relleno,relleno,relleno,relleno,relleno,relleno,relleno,relleno,relleno,relleno,relleno,relleno,relleno,relleno,relleno,relleno,relleno,relleno,relleno,relleno,relleno,relleno,relleno,relleno,relleno,relleno,relleno,relleno]

  	#P_Tipo1_Mos9 = [WP1_Mos9_T1_p,WP2_Mos9_T1_p,WP3_Mos9_T1_p,WP4_Mos9_T1_p,WP5_Mos9_T1_p,WP6_Mos9_T1_p,WP7_Mos9_T1_p,WP8_Mos9_T1_p,WP9_Mos9_T1_p,WP10_Mos9_T1_p,relleno,relleno,relleno,relleno,relleno,relleno,relleno,relleno,relleno,relleno,relleno,relleno,relleno,relleno,relleno,relleno,relleno,relleno,relleno,relleno,relleno,relleno,relleno,relleno,relleno,relleno,relleno,relleno,relleno,relleno]
  	#P_Tipo2_Mos9 = [WP1_Mos9_T2_p,WP2_Mos9_T2_p,WP3_Mos9_T2_p,WP4_Mos9_T2_p,WP5_Mos9_T2_p,WP6_Mos9_T2_p,WP7_Mos9_T2_p,WP8_Mos9_T2_p,WP9_Mos9_T2_p,WP10_Mos9_T2_p,relleno,relleno,relleno,relleno,relleno,relleno,relleno,relleno,relleno,relleno,relleno,relleno,relleno,relleno,relleno,relleno,relleno,relleno,relleno,relleno,relleno,relleno,relleno,relleno,relleno,relleno,relleno,relleno,relleno,relleno]

  	#P_Tipo1_Mos10 = [WP1_Mos10_T1_p,WP2_Mos10_T1_p,WP3_Mos10_T1_p,WP4_Mos10_T1_p,WP5_Mos10_T1_p,WP6_Mos10_T1_p,WP7_Mos10_T1_p,WP8_Mos10_T1_p,WP9_Mos10_T1_p,WP10_Mos10_T1_p,relleno,relleno,relleno,relleno,relleno,relleno,relleno,relleno,relleno,relleno,relleno,relleno,relleno,relleno,relleno,relleno,relleno,relleno,relleno,relleno,relleno,relleno,relleno,relleno,relleno,relleno,relleno,relleno,relleno,relleno]
  	#P_Tipo2_Mos10 = [WP1_Mos10_T2_p,WP2_Mos10_T2_p,WP3_Mos10_T2_p,WP4_Mos10_T2_p,WP5_Mos10_T2_p,WP6_Mos10_T2_p,WP7_Mos10_T2_p,WP8_Mos10_T2_p,WP9_Mos10_T2_p,WP10_Mos10_T2_p,relleno,relleno,relleno,relleno,relleno,relleno,relleno,relleno,relleno,relleno,relleno,relleno,relleno,relleno,relleno,relleno,relleno,relleno,relleno,relleno,relleno,relleno,relleno,relleno,relleno,relleno,relleno,relleno,relleno,relleno]

  	#P_Tipo1_Mos11 = [WP1_Mos11_T1_p,WP2_Mos11_T1_p,WP3_Mos11_T1_p,WP4_Mos11_T1_p,WP5_Mos11_T1_p,WP6_Mos11_T1_p,WP7_Mos11_T1_p,WP8_Mos11_T1_p,WP9_Mos11_T1_p,WP10_Mos11_T1_p,relleno,relleno,relleno,relleno,relleno,relleno,relleno,relleno,relleno,relleno,relleno,relleno,relleno,relleno,relleno,relleno,relleno,relleno,relleno,relleno,relleno,relleno,relleno,relleno,relleno,relleno,relleno,relleno,relleno,relleno]
  	#P_Tipo2_Mos11 = [WP1_Mos11_T2_p,WP2_Mos11_T2_p,WP3_Mos11_T2_p,WP4_Mos11_T2_p,WP5_Mos11_T2_p,WP6_Mos11_T2_p,WP7_Mos11_T2_p,WP8_Mos11_T2_p,WP9_Mos11_T2_p,WP10_Mos11_T2_p,relleno,relleno,relleno,relleno,relleno,relleno,relleno,relleno,relleno,relleno,relleno,relleno,relleno,relleno,relleno,relleno,relleno,relleno,relleno,relleno,relleno,relleno,relleno,relleno,relleno,relleno,relleno,relleno,relleno,relleno]

  	#P_Tipo1_Mos12 = [WP1_Mos12_T1_p,WP2_Mos12_T1_p,WP3_Mos12_T1_p,WP4_Mos12_T1_p,WP5_Mos12_T1_p,WP6_Mos12_T1_p,WP7_Mos12_T1_p,WP8_Mos12_T1_p,WP9_Mos12_T1_p,WP10_Mos12_T1_p,WP11_Mos12_T1_p,WP12_Mos12_T1_p,WP13_Mos12_T1_p,WP14_Mos12_T1_p,WP15_Mos12_T1_p,WP16_Mos12_T1_p,WP17_Mos12_T1_p,WP18_Mos12_T1_p,WP19_Mos12_T1_p,WP20_Mos12_T1_p,WP21_Mos12_T1_p,WP22_Mos12_T1_p,WP23_Mos12_T1_p,WP24_Mos12_T1_p,WP25_Mos12_T1_p,WP26_Mos12_T1_p,WP27_Mos12_T1_p,WP28_Mos12_T1_p,WP29_Mos12_T1_p,WP30_Mos12_T1_p,WP31_Mos12_T1_p,WP32_Mos12_T1_p,relleno,relleno,relleno,relleno,relleno,relleno,relleno,relleno]
  	#P_Tipo2_Mos12 = [WP1_Mos12_T2_p,WP2_Mos12_T2_p,WP3_Mos12_T2_p,WP4_Mos12_T2_p,WP5_Mos12_T2_p,WP6_Mos12_T2_p,WP7_Mos12_T2_p,WP8_Mos12_T2_p,WP9_Mos12_T2_p,WP10_Mos12_T2_p,WP11_Mos12_T2_p,WP12_Mos12_T2_p,WP13_Mos12_T2_p,WP14_Mos12_T2_p,WP15_Mos12_T2_p,WP16_Mos12_T2_p,WP17_Mos12_T2_p,WP18_Mos12_T2_p,WP19_Mos12_T2_p,WP20_Mos12_T2_p,WP21_Mos12_T2_p,WP22_Mos12_T2_p,WP23_Mos12_T2_p,WP24_Mos12_T2_p,WP25_Mos12_T2_p,WP26_Mos12_T2_p,WP27_Mos12_T2_p,WP28_Mos12_T2_p,WP29_Mos12_T2_p,WP30_Mos12_T2_p,WP31_Mos12_T2_p,WP32_Mos12_T2_p,relleno,relleno,relleno,relleno,relleno,relleno,relleno,relleno]


  	PuntosCogida = [PCogida_P1_p,PCogida_P1_p,PCogida_P1_p,relleno,relleno,relleno,relleno,relleno,relleno,relleno,relleno,relleno,relleno,relleno,relleno]
                 PuntosCogida[0] = PCogida_P1_p


      local i = 0
      while i < 40:

          P_Tipo1_Mos1[i] = pose_trans(Pbf,P_Tipo1_Mos1[i])
          P_Tipo2_Mos1[i] = pose_trans(Pbf,P_Tipo2_Mos1[i])

          #P_Tipo1_Mos2[i] = pose_trans(Pbf,P_Tipo1_Mos2[i])
          #P_Tipo2_Mos2[i] = pose_trans(Pbf,P_Tipo2_Mos2[i])

          #P_Tipo1_Mos3[i] = pose_trans(Pbf,P_Tipo1_Mos3[i])
          #P_Tipo2_Mos3[i] = pose_trans(Pbf,P_Tipo2_Mos3[i])

          #P_Tipo1_Mos4[i] = pose_trans(Pbf,P_Tipo1_Mos4[i])
          #P_Tipo2_Mos4[i] = pose_trans(Pbf,P_Tipo2_Mos4[i])

          #P_Tipo1_Mos5[i] = pose_trans(Pbf,P_Tipo1_Mos5[i])
          #P_Tipo2_Mos5[i] = pose_trans(Pbf,P_Tipo2_Mos5[i])

          #P_Tipo1_Mos6[i] = pose_trans(Pbf,P_Tipo1_Mos6[i])
          #P_Tipo2_Mos6[i] = pose_trans(Pbf,P_Tipo2_Mos6[i])

          #P_Tipo1_Mos7[i] = pose_trans(Pbf,P_Tipo1_Mos7[i])
          #P_Tipo2_Mos7[i] = pose_trans(Pbf,P_Tipo2_Mos7[i])

          #P_Tipo1_Mos8[i] = pose_trans(Pbf,P_Tipo1_Mos8[i])
          #P_Tipo2_Mos8[i] = pose_trans(Pbf,P_Tipo2_Mos8[i])

          #P_Tipo1_Mos9[i] = pose_trans(Pbf,P_Tipo1_Mos9[i])
          #P_Tipo2_Mos9[i] = pose_trans(Pbf,P_Tipo2_Mos9[i])

          #P_Tipo1_Mos10[i] = pose_trans(Pbf,P_Tipo1_Mos10[i])
          #P_Tipo2_Mos10[i] = pose_trans(Pbf,P_Tipo2_Mos10[i])

          #P_Tipo1_Mos11[i] = pose_trans(Pbf,P_Tipo1_Mos11[i])
          #P_Tipo2_Mos11[i] = pose_trans(Pbf,P_Tipo2_Mos11[i])

          #P_Tipo1_Mos12[i] = pose_trans(Pbf,P_Tipo1_Mos12[i])
          #P_Tipo2_Mos12[i] = pose_trans(Pbf,P_Tipo2_Mos12[i])

          i = i + 1
      end

      reset_puntos = False
  end
  $ 4 "Script: InitReg.script"
  #Para enviar a la pantalla los valores nada más inicializar
  write_output_boolean_register(0,LineaHabilitada[0])
  write_output_boolean_register(1,LineaHabilitada[1])
  $ 5 "Script: Funciones.script"
  #Función para la creación de un popup informativo que desaparece (y opcionalmente se aborta el Programa_1) tras un tiempo de espera
  def pop_up(mensaje, tiempo_espera, aborto):
  	socket_open("127.0.0.1",29999,"internal")
  	socket_send_string("popup " + mensaje, "internal")
  	socket_send_byte(10,"internal")

  	sleep(tiempo_espera)

  	socket_send_string("close popup", "internal")
  	socket_send_byte(10,"internal")

  	socket_close("internal")

  	if aborto == True:
  		halt
  	end

  end

  #Función que se usa para actualizar el TCP cuando hay cambio de peso, coordenadas o cog
  def setTCP(tool):

  	tool_tcp = p[tool[0]/1000, tool[1]/1000, tool[2]/1000, tool[3], tool[4], tool[5]]
  	mass = tool[6]/1000
  	cog = [tool[7]/1000, tool[8]/1000, tool[9]/1000]

  	set_tcp(tool_tcp)
  	set_payload(mass, cog)

  end


  #Funciones de movimiento respecto a un plano
  def MoveLTrans(p_destino, WorkObject, aceleracion, velocidad, tiempo, contorneo):

  	#El WorkObject debe tener la misma orientacion en Z que el TCP que vamos a utilizar
  	p_trans=pose_trans(WorkObject,p_destino)
  	movel(p_trans,aceleracion,velocidad,tiempo, contorneo)

  end


  def MoveJTrans(p_destino, WorkObject, aceleracion, velocidad, tiempo, contorneo):

  	#El WorkObject debe tener la misma orientacion en Z que el TCP que vamos a utilizar
  	p_trans=pose_trans(WorkObject,p_destino)
  	movej(p_trans,aceleracion,velocidad, tiempo, contorneo)

  end


  def MovePTrans(p_destino, WorkObject, aceleracion, velocidad, tiempo, contorneo):

  	#El WorkObject debe tener la misma orientacion en Z que el TCP que vamos a utilizar
  	p_trans=pose_trans(WorkObject,p_destino)
  	movep(p_trans,aceleracion,velocidad, tiempo, contorneo)

  end


  #Función de palet completo
  def palet_completo(lin):

  	PalletEnd[lin] = True
  	NCapaAct[lin] = 1
  	NPrdAct[lin] = 1
  	NMovAct[lin] = 1
  	NPaletAct = NPaletAct + 1
  	NPaletTot = NPaletTot + 1

  	if NPaletTot == 800000:
  		NPaletTot = 1
  	end

  	if NPaletAct == 800000:
  		NPaletAct = 1
  	end

  	pos_subida[lin] = 0
  	pos_bajada[lin] = 0

  end
  $ 6 "Script: FiltroES.script"
  #Creacion de variables de trabajo entrada (las que filtro)
  global FT1_work = False
  global FT2_work = False
  global AVISO_SAI = False     #Cambio RGR 23/11/2022, nueva variable#
  global FT4_work = False
  global FT5_work = False
  global QM1_work = False
  global VF1_work = False
  global QM2_work = False
  global VF2_work = False

  global parpadeo = False

  #Definición TEMPORIZADORES

  #tON
  global temp_tON_FT1=0
  global temp_tON_FT2=0
  global temp_tON_AVISO_SAI=0		#Cambio RGR 23/11/2022, nueva variable#
  global temp_tON_FT4=0
  global temp_tON_FT5=0
  global temp_tON_QM1=0
  global temp_tON_VF1=0
  global temp_tON_QM2=0
  global temp_tON_VF2=0


  #tOFF
  global temp_tOFF_FT1=0
  global temp_tOFF_FT2=0
  global temp_tOFF_AVISO_SAI=0				#Cambio RGR 23/11/2022, nueva variable#
  global temp_tOFF_FT4=0
  global temp_tOFF_FT5=0
  global temp_tOFF_QM1=0
  global temp_tOFF_VF1=0
  global temp_tOFF_QM2=0
  global temp_tOFF_VF2=0


  #Balizas
  global temp_parpadeo = 0

  #Alarmas

  global temp_alarmas = [0,0,0,0,0,0,0,0,0,0,0,0,0,0,0,0,0,0,0,0,0,0,0,0,0,0,0,0,0,0,0,0,0,0,0,0,0,0,0,0,0,0,0,0,0,0,0,0,0,0]

  #Contador TEMPORIZADORES
  #FILTRADO ENTRADAS
  thread thread_filtrado():
  	while(True):

  	  #Lectura de entradas
  	  FT1_work = not(get_standard_digital_in(0))
  	  FT2_work = not(get_standard_digital_in(1))
  	  AVISO_SAI = get_standard_digital_in(2)
  	  FT4_work = not(get_standard_digital_in(3))
  	  FT5_work = get_standard_digital_in(4)
  	  QM1_work = not(get_standard_digital_in(7))
  	  VF1_work = get_configurable_digital_in(0)
  	  QM2_work = not(get_configurable_digital_in(6))
  	  VF2_work = get_configurable_digital_in(7)
  	  iVAC1 = get_tool_digital_in(0)
  	  iVAC2 = get_tool_digital_in(1)


  	  #FT1
  	  if (FT1_work):
  		temp_tON_FT1 = temp_tON_FT1 + retraso
  		temp_tOFF_FT1 = 0
  	  else:
  		temp_tOFF_FT1 = temp_tOFF_FT1 + retraso
  		temp_tON_FT1 = 0
  	  end

  	  if (temp_tON_FT1 > tON_FT1):
  		iFT1 =  True
  		temp_tON_FT1 = 0
  	  end

  	  if (temp_tOFF_FT1 > tOFF_FT1):
  		iFT1 =  False
  		temp_tOFF_FT1 = 0
  	  end

  	  #FT2
  	  if (FT2_work):
  		temp_tON_FT2 = temp_tON_FT2 + retraso
  		temp_tOFF_FT2 = 0
  	  else:
  		temp_tOFF_FT2 = temp_tOFF_FT2 + retraso
  		temp_tON_FT2 = 0
  	  end

  	  if (temp_tON_FT2 > tON_FT2):
  		iFT2 =  True
  		temp_tON_FT2 = 0
  	  end

  	  if (temp_tOFF_FT2 > tOFF_FT2):
  		iFT2 =  False
  		temp_tOFF_FT2 = 0
  	  end

  	  #Aviso_SAI
  	  if (AVISO_SAI):							#Cambio RGR 23/11/2022, nuevo#
  		temp_tON_AVISO_SAI = temp_tON_AVISO_SAI + retraso	#Cambio RGR 23/11/2022, nuevo#
  		temp_tOFF_AVISO_SAI = 0					#Cambio RGR 23/11/2022, nuevo#
  	  else:								#Cambio RGR 23/11/2022, nuevo#
  		temp_tOFF_AVISO_SAI = temp_tOFF_AVISO_SAI + retraso	#Cambio RGR 23/11/2022, nuevo#
  		temp_tON_AVISO_SAI = 0					#Cambio RGR 23/11/2022, nuevo#
  	  end								#Cambio RGR 23/11/2022, nuevo#

  	if (temp_tON_AVISO_SAI > tON_AVISO_SAI):				#Cambio RGR 23/11/2022, nuevo#
  		iAVISO_SAI =  True					#Cambio RGR 23/11/2022, nuevo#
  		temp_tON_AVISO_SAI = 0					#Cambio RGR 23/11/2022, nuevo#
  	  end								#Cambio RGR 23/11/2022, nuevo#

  	  if (temp_tOFF_AVISO_SAI > tOFF_AVISO_SAI):			#Cambio RGR 23/11/2022, nuevo#
  		iAVISO_SAI =  False					#Cambio RGR 23/11/2022, nuevo#
  		temp_tOFF_AVISO_SAI = 0					#Cambio RGR 23/11/2022, nuevo#
  	  end								#Cambio RGR 23/11/2022, nuevo#

  	  #FT4
  	  if (FT4_work):
  		temp_tON_FT4 = temp_tON_FT4 + retraso
  		temp_tOFF_FT4 = 0
  	  else:
  		temp_tOFF_FT4 = temp_tOFF_FT4 + retraso
  		temp_tON_FT4 = 0
  	  end

  	  if (temp_tON_FT4 > tON_FT4):
  		iFT4 =  True
  		temp_tON_FT4 = 0
  	  end

  	  if (temp_tOFF_FT4 > tOFF_FT4):
  		iFT4 =  False
  		temp_tOFF_FT4 = 0
  	  end

  	  #FT5
  	  if (FT5_work):
  		temp_tON_FT5 = temp_tON_FT5 + retraso
  		temp_tOFF_FT5 = 0
  	  else:
  		temp_tOFF_FT5 = temp_tOFF_FT5 + retraso
  		#temp_tON_FT5 = 0
  	  end

  	  if (temp_tON_FT5 > tON_FT5):
  		iFT5 =  True
  		temp_tON_FT5 = 0
  	  end

  	  if (temp_tOFF_FT5 > tOFF_FT5):
  		iFT5 =  False
  		temp_tOFF_FT5 = 0
  	  end

  	  #QM1
  	  if (QM1_work):
  		temp_tON_QM1 = temp_tON_QM1 + retraso
  		temp_tOFF_QM1 = 0
  	  else:
  		temp_tOFF_QM1 = temp_tOFF_QM1 + retraso
  		temp_tON_QM1 = 0
  	  end

  	  if (temp_tON_QM1 > tON_QM1):
  		iQM1 =  True
  		temp_tON_QM1 = 0
  	  end

  	  if (temp_tOFF_QM1 > tOFF_QM1):
  		iQM1 =  False
  		temp_tOFF_QM1 = 0
  	  end

  	  #VF1
  	  if (VF1_work):
  		temp_tON_VF1 = temp_tON_VF1 + retraso
  		temp_tOFF_VF1 = 0
  	  else:
  		temp_tOFF_VF1 = temp_tOFF_VF1 + retraso
  		temp_tON_VF1 = 0
  	  end

  	  if (temp_tON_VF1 > tON_VF1):
  		iVF1 =  True
  		temp_tON_VF1 = 0
  	  end

  	  if (temp_tOFF_VF1 > tOFF_VF1):
  		iVF1 =  False
  		temp_tOFF_VF1 = 0
  	  end

  	  #QM2
  	  if (QM2_work):
  		temp_tON_QM2 = temp_tON_QM2 + retraso
  		temp_tOFF_QM2 = 0
  	  else:
  		temp_tOFF_QM2 = temp_tOFF_QM2 + retraso
  		temp_tON_QM2 = 0
  	  end

  	  if (temp_tON_QM2 > tON_QM2):
  		iQM2 =  True
  		temp_tON_QM2 = 0
  	  end

  	  if (temp_tOFF_QM2 > tOFF_QM2):
  		iQM2 =  False
  		temp_tOFF_QM2 = 0
  	  end

  	  #VF2
  	  if (VF2_work):
  		temp_tON_VF2 = temp_tON_VF2 + retraso
  		temp_tOFF_VF2 = 0
  	  else:
  		temp_tOFF_VF2 = temp_tOFF_VF2 + retraso
  		temp_tON_VF2 = 0
  	  end

  	  if (temp_tON_VF2 > tON_VF2):
  		iVF2 =  True
  		temp_tON_VF2 = 0
  	  end

  	  if (temp_tOFF_VF2 > tOFF_VF2):
  		iVF2 =  False
  		temp_tOFF_VF2 = 0
  	  end

  	  #parpadeo
  	  temp_parpadeo = temp_parpadeo + retraso
  	  if (temp_parpadeo > 1.0):
  		parpadeo = not(parpadeo)
  		temp_parpadeo = 0
  	  end

  	  #ALARMAS

  	  #Alarma vacío
  #	  if (oEV4 == False):
  #		temp_alarmas[0] = temp_alarmas[0] + retraso
  #		if(temp_alarmas[0] > 10):
  #			if(iRD2 == False):
  #				AlarmaVacio = True
  #			else:
  #				temp_alarmas[0] = 0
  #			end
  #		end
  #	  else:
  #		temp_alarmas[0] = 0
  #	  end

  	  #Alarma VF2
  	  if (oM2 == True):
  		temp_alarmas[1] = temp_alarmas[1] + retraso
          		if (temp_alarmas[1] > 3):
  			if(iVF2 == False):
  				AlarmaVF2 = True

  			else:
  				temp_alarmas[1] = 0
  			end
  		end
  	  else:
  		temp_alarmas[1] = 0
        	end

  	if (oM2 == False):
  		temp_alarmas[2] = temp_alarmas[2] + retraso
  	    	if (temp_alarmas[2] > 3):
  			if(iVF2 == True):
  				AlarmaVF2 = True

  			else:
  				temp_alarmas[2] = 0
  			end
  		end
  	else:
  		temp_alarmas[2] = 0
        	end

  	  #Alarma QM2
  	  if (iQM2 == True):
  		AlarmaQM2 = True
  	  end

  	  #ACTUALIZACIÓN REGISTROS

  	  #Sólo lectura Java --> Robot
  	  LineaHabilitada[0] = read_output_boolean_register(0)
  	  LineaHabilitada[1] = read_output_boolean_register(1)
  	  DescargarPal[0] = read_output_boolean_register(2)
  	  DescargarPal[1] = read_output_boolean_register(3)
  	  ResetSec = read_output_boolean_register(4)
  	  CambioPrograma = read_output_boolean_register(5)
  	  CambiosAvanzados = read_output_boolean_register(6)
  	  ResetAlarmas = read_output_boolean_register(16)
  	  #ProgRunning = read_output_boolean_register(15)

  	  #Solo lectura Robot --> Java
  	  #Bool
  	  write_output_boolean_register(7,PermisoBotones)
  	  write_output_boolean_register(8,PalletReady[0])
  	  write_output_boolean_register(9,PalletReady[1])
  	  write_output_boolean_register(10,PalletEnd[0])
  	  write_output_boolean_register(11,PalletEnd[1])
  	  write_output_boolean_register(12,ProdListo)
  	  write_output_boolean_register(13,ManoConProd)
  	  write_output_boolean_register(14,Rec_CapasTrab[Programa_1-1])
  	  #recordar que ProgRunning se configura en instalación

  	  write_output_boolean_register(17,Aviso)
  	  write_output_boolean_register(18,AvisoPaletCompletoL1)
  	  write_output_boolean_register(19,AvisoPaletCompletoL2)
  	  write_output_boolean_register(20,AvisoL1Deshab)
  	  write_output_boolean_register(21,AvisoL2Deshab)
  	  write_output_boolean_register(22,AvisoPaletL1)
  	  write_output_boolean_register(23,AvisoPaletL2)
  	  write_output_boolean_register(25,Alarma)
  	  write_output_boolean_register(26,AlarmaVacio)
  	  write_output_boolean_register(33,AlarmaVF2)
  	  write_output_boolean_register(34,AlarmaQM2)
  	  write_output_boolean_register(35,iAVISO_SAI)

  	  write_output_boolean_register(36,ManoConCarton)
  	  write_output_boolean_register(37,CartonBase[0])
  	  write_output_boolean_register(38,CartonBase[1])
  	  write_output_boolean_register(39,PonerCarton[0])
  	  write_output_boolean_register(40,PonerCarton[1])


  	  write_output_boolean_register(92,iFT1)
  	  write_output_boolean_register(93,iFT2)
  	  write_output_boolean_register(95,iFT4)
  	  write_output_boolean_register(96,iFT5)

  	  #write_output_boolean_register(99,iQM1)
  	  #write_output_boolean_register(100,iVF1)
  	  write_output_boolean_register(106,iQM2)
  	  write_output_boolean_register(107,iVF2)

  	  write_output_boolean_register(110,oEV1)
  	  #write_output_boolean_register(111,oEV2)
  	  write_output_boolean_register(112,oB1V)
  	  write_output_boolean_register(113,oB1R)
  	  write_output_boolean_register(114,oB2V)
  	  write_output_boolean_register(115,oB2R)
  	  #write_output_boolean_register(116,oEV3)
  	  write_output_boolean_register(117,oEV4)
  	  #write_output_boolean_register(118,oEV5)
  	  #write_output_boolean_register(119,oM1)
  	  write_output_boolean_register(120,oM2)
  	  #write_output_boolean_register(121,oRP_ME)



  	  #Integer variables enteras
  	  write_output_integer_register(32,NCapaAct[0])
  	  write_output_integer_register(33,NCapaAct[1])
  	  write_output_integer_register(34,NMovAct[0])
  	  write_output_integer_register(35,NMovAct[1])
  	  write_output_integer_register(36,PrdsReq)
  	  write_output_integer_register(37,ContPrd)
  	  write_output_integer_register(38,NPaletAct)
  	  write_output_integer_register(39,NPaletTot)
  	  write_output_integer_register(40,linea)
  	  write_output_integer_register(41,Programa_1)
  	  write_output_integer_register(42,Rec_Mosaico[Programa_1-1])
  	  write_output_integer_register(43,Rec_LargoPrd[Programa_1-1])
  	  write_output_integer_register(44,Rec_AnchoPrd[Programa_1-1])
  	  write_output_integer_register(45,Rec_NCapasTot[Programa_1-1])
  	  write_output_integer_register(46,Rec_NMovsCapa[Programa_1-1])
  	  write_output_integer_register(47,StepCode)

  	  #Float
  	  write_output_float_register(46,Rec_AltoPrd[Programa_1-1])
  	  write_output_float_register(47,Rec_PesoPrd[Programa_1-1])

  	  #ACTUALIZACIÓN SALIDAS
  	  # 'EV1'
  	  set_standard_digital_out(0,oEV1)
  	  # 'EV2'
  	  set_standard_digital_out(1,oEV2)
  	  # 'B1V'
  	  set_standard_digital_out(2,oB1V)
  	  # 'B1R'
  	  set_standard_digital_out(3,oB1R)
  	  # 'B2V'
  	  set_standard_digital_out(4,oB2V)
  	  # 'B2R'
  	  set_standard_digital_out(5,oB2R)
  	  # 'EV3'
  	  #set_standard_digital_out(6,oEV3)
  	  # 'EV4'
  	  set_standard_digital_out(7,oEV4)
  	  # 'EV5'
  	  set_configurable_digital_out(0,oEV5)
  	  # 'M1'
  	  set_configurable_digital_out(1,oM1)
  	  # 'M2'
        	  set_configurable_digital_out(2,oM2)
  	  # 'RP_ME'
  	  set_configurable_digital_out(3,oRP_ME)

  	  # 'VELM1'
  	  set_standard_analog_out(0,oVELM1)
  	  # 'VELM2'
  	  set_standard_analog_out(1,oVELM2)


  	  sleep(retraso)

  	end
  end
  run thread_filtrado()



  $ 7 "Call Inicializacion"
  Inicializacion()
  $ 8 "Call CargarDatos"
  CargarDatos()
  $ 9 "Script: Calculos_perch.script"
  local j = 0

  yPPerchDejada_min_array = [1,1]
  yPPerchDejada_max_array = [0,0]
  xPPerchDejada_array = [1,1]

  local punto_aux = P_Tipo1[j]
  yPPerchDejada_min_array[0] = punto_aux[1]
  yPPerchDejada_max_array[0] = punto_aux[1]
  xPPerchDejada_array[0] = punto_aux[0]

   while j < Rec_NMovsCapa[Programa_1-1]:
   #while j < 15:
      if punto_aux[1] < yPPerchDejada_min_array[0]:
          yPPerchDejada_min_array[0] = punto_aux[1]
      end
      if punto_aux[1] > yPPerchDejada_max_array[0]:
          yPPerchDejada_max_array[0] = punto_aux[1]
      end
      if punto_aux[0] < xPPerchDejada_array[0]:
         xPPerchDejada_array[0] = punto_aux[0]
      end
      j = j + 1
      punto_aux = P_Tipo1[j]
      sleep(0.01)
  end

  if Rec_CapasTrab[Programa_1-1]:

  	j = 0

  	punto_aux = P_Tipo2[j]
  	yPPerchDejada_min_array[1] = punto_aux[1]
  	yPPerchDejada_max_array[1] = punto_aux[1]
  	xPPerchDejada_array[1] = punto_aux[0]

  	while j < Rec_NMovsCapa[Programa_1-1]:
  #while j < 15:
      		if punto_aux[1] < yPPerchDejada_min_array[1]:
          			yPPerchDejada_min_array[1] = punto_aux[1]
      		end
      		if punto_aux[1] > yPPerchDejada_max_array[1]:
          			yPPerchDejada_max_array[1] = punto_aux[1]
      		end
      		if punto_aux[0] < xPPerchDejada_array[1]:
         			xPPerchDejada_array[1] = punto_aux[0]
      		end
      		j = j + 1
      		punto_aux = P_Tipo2[j]
      		sleep(0.01)
  	end

  end

  if yPPerchDejada_min_array[1]<yPPerchDejada_min_array[0]:
  	global yPPerchDejada_min = yPPerchDejada_min_array[1]
  else:
  	global yPPerchDejada_min = yPPerchDejada_min_array[0]
  end

  if yPPerchDejada_max_array[1]>yPPerchDejada_max_array[0]:
  	global yPPerchDejada_max = yPPerchDejada_max_array[1]
  else:
  	global yPPerchDejada_max = yPPerchDejada_max_array[0]
  end

  if xPPerchDejada_array[1]<xPPerchDejada_array[0]:
  	global xPPerchDejada = xPPerchDejada_array[1]
  else:
  	global xPPerchDejada = xPPerchDejada_array[0]
  end


  if Rec_CapasTrab[Programa_1-1] == True:
  	Rec_TipoCapa = [1, 2, 1, 2, 1, 2, 1, 2, 1, 2, 1, 2, 1, 2, 1, 2, 1, 2, 1, 2, 1, 2, 1, 2, 1, 2, 1, 2, 1, 2]

  else:
  	Rec_TipoCapa = [1,1,1,1,1,1,1,1,1,1,1,1,1,1,1,1,1,1,1,1,1,1,1,1,1,1,1,1,1,1]
  end


  #Dónde poner cartón en función del Programa_1
  #if Programa_1 == 12:
  	#Rec_Carton = #[True,False,False,True,False,False,True,False,False,True,False,False,True,False,False,True,False,False,True,False,False,True,False,False,True,False,False,True,False,False]

  #else:
  	#Rec_Carton = #[False,False,False,False,False,False,False,False,False,False,False,False,False,False,False,False,False,False,False,False,False,False,False,False,False,False,False,False,False,False]
  #end
  $ 335 "Thread_1"
  thread Thread_1():
    while (True):
      $ 336 "Thread_ProductoListo"
      $ 337 "If iFT4"
      if (iFT4):
        $ 338 "ProdListo = True"
        ProdListo = True
        $ 339 "ContPrd=1"
        ContPrd=1
      else:
        $ 341 "Else" "noBreak"
        $ 342 "ProdListo = False"
        ProdListo = False
        $ 343 "ContPrd=0"
        ContPrd=0
      end
      $ 344 "Thread_LineaPreparada"
      $ 345 "If iFT1"
      if (iFT1):
        $ 346 "PalletReady[0] =  True "
        PalletReady[0] =   True
      else:
        $ 347 "Else" "noBreak"
        $ 348 "PalletReady[0] =  False "
        PalletReady[0] =   False
        $ 349 "PalletEnd[0] =  False "
        PalletEnd[0] =   False
      end
      $ 350 "If iFT2"
      if (iFT2):
        $ 351 "PalletReady[1] =  True "
        PalletReady[1] =   True
      else:
        $ 352 "Else" "noBreak"
        $ 353 "PalletReady[1] =  False "
        PalletReady[1] =   False
        $ 354 "PalletEnd[1] =  False "
        PalletEnd[1] =   False
      end
      $ 355 "PalletOk[1]=PalletReady[1]  and  PalletEnd[1]≟ False "
      PalletOk[1]=PalletReady[1]   and   PalletEnd[1] ==   False
      $ 356 "PalletOk[0]=PalletReady[0]  and  PalletEnd[0]≟ False "
      PalletOk[0]=PalletReady[0]   and   PalletEnd[0] ==   False
      $ 357 "LineaPreparada[0]=PalletOk[0] and LineaHabilitada[0] and (ProdListo or (not(CartonBase[0]) and NCapaAct[0]≟1  and NMovAct[0]≟1 and Rec_Carton[0])  or PonerCarton[0])"
      LineaPreparada[0]=PalletOk[0]  and  LineaHabilitada[0]  and  (ProdListo or (not(CartonBase[0])  and  NCapaAct[0] == 1  and NMovAct[0] == 1 and Rec_Carton[0])   or  PonerCarton[0])
      $ 358 "LineaPreparada[1]=PalletOk[1] and LineaHabilitada[1] and (ProdListo or (not(CartonBase[1]) and NCapaAct[1]≟1 and NMovAct[1] ≟ 1 and Rec_Carton[0])  or  PonerCarton[1])"
      LineaPreparada[1]=PalletOk[1]  and  LineaHabilitada[1]  and  (ProdListo or (not(CartonBase[1])  and  NCapaAct[1] == 1 and NMovAct[1]  ==  1 and Rec_Carton[0])   or   PonerCarton[1])
      $ 359 "Thread_DescargaPalet y Reset Secuencia"
      $ 360 "If PermisoBotones and DescargarPal[0]"
      if (PermisoBotones  and  DescargarPal[0]):
        $ 361 "palet_completo(0)"
        palet_completo(0)
        $ 362 "write_output_boolean_register(2,False)"
        write_output_boolean_register(2,False)
        $ 363 "'DescargarPal[0] = False'"
        # 'DescargarPal[0] = False'
        $ 364 "CartonBase[0] = False"
        CartonBase[0] = False
      end
      $ 366 "If PermisoBotones and DescargarPal[1]"
      if (PermisoBotones  and  DescargarPal[1]):
        $ 367 "palet_completo(1)"
        palet_completo(1)
        $ 368 "write_output_boolean_register(3,False)"
        write_output_boolean_register(3,False)
        $ 369 "'DescargarPal[1] = False'"
        # 'DescargarPal[1] = False'
        $ 370 "CartonBase[1] = False"
        CartonBase[1] = False
      end
      $ 372 "If PermisoBotones and ResetSec"
      if (PermisoBotones  and  ResetSec):
        $ 373 "ProdListo = False"
        ProdListo = False
        $ 374 "M_PL =  False "
        M_PL =   False
        $ 375 "write_output_boolean_register(4,False)"
        write_output_boolean_register(4,False)
        $ 376 "'ResetSec = False'"
        # 'ResetSec = False'
        $ 377 "ContPrd = 0"
        ContPrd = 0
      end
      $ 378 "If Rec_Cogida2en2[Programa_1-1]≟ False "
      if (Rec_Cogida2en2[Programa_1-1] ==   False  ):
        $ 379 "PrdsReq = 1"
        PrdsReq = 1
      else:
        $ 380 "Else" "noBreak"
        $ 381 "PrdsReq = 2"
        PrdsReq = 2
      end
      $ 382 "Thread_permisos"
      $ 383 "If LineaHabilitada[0] ≟ False  and LineaHabilitada[1]≟ False  and StepCode≟4"
      if (LineaHabilitada[0]  ==   False    and  LineaHabilitada[1] ==   False    and  StepCode == 4):
        $ 384 "PermisoBotones = True"
        PermisoBotones = True
      else:
        $ 385 "Else" "noBreak"
        $ 386 "PermisoBotones = False"
        PermisoBotones = False
      end
      $ 387 "Thread_motor"
      $ 390 "If StepCode≤3  and StepCode≥13"
      if (StepCode <= 3   and  StepCode >= 13):
        $ 391 "oM2 = False "
        oM2 =  False
      else:
        $ 392 "Else" "noBreak"
        $ 393 "oM2 = True "
        oM2 =  True
      end
      $ 394 "Thread_Baliza1"
      $ 395 "If PalletEnd[0]"
      if (PalletEnd[0]):
        $ 396 "oB1R = True "
        oB1R =  True
        $ 397 "oB1V = False "
        oB1V =  False
      end
      $ 398 "If (LineaHabilitada[0]≟ False  or PalletReady[0]≟ False ) and PalletEnd[0]≟ False "
      if ((LineaHabilitada[0] ==   False    or  PalletReady[0] ==   False  )  and  PalletEnd[0] ==   False  ):
        $ 399 "oB1R =parpadeo"
        oB1R =parpadeo
        $ 400 "oB1V = False "
        oB1V =  False
      end
      $ 401 "If LineaHabilitada[0] and PalletReady[0] and linea≠1 and PalletEnd[0]≟ False "
      if (LineaHabilitada[0]  and  PalletReady[0]  and  linea != 1  and  PalletEnd[0] ==   False  ):
        $ 402 "oB1V =parpadeo"
        oB1V =parpadeo
        $ 403 "oB1R = False "
        oB1R =  False
      end
      $ 404 "If LineaHabilitada[0] and PalletReady[0] and linea≟1 and PalletEnd[0]≟ False "
      if (LineaHabilitada[0]  and  PalletReady[0]  and  linea == 1  and  PalletEnd[0] ==   False  ):
        $ 405 "oB1V = True "
        oB1V =  True
        $ 406 "oB1R = False "
        oB1R =  False
      end
      $ 407 "Thread_Baliza2"
      $ 408 "If PalletEnd[1]"
      if (PalletEnd[1]):
        $ 409 "oB2R = True "
        oB2R =  True
        $ 410 "oB2V = False "
        oB2V =  False
      end
      $ 411 "If (LineaHabilitada[1]≟ False  or PalletReady[1]≟ False ) and PalletEnd[1]≟ False "
      if ((LineaHabilitada[1] ==   False    or  PalletReady[1] ==   False  )  and  PalletEnd[1] ==   False  ):
        $ 412 "oB2R =parpadeo"
        oB2R =parpadeo
        $ 413 "oB2V = False "
        oB2V =  False
      end
      $ 414 "If LineaHabilitada[1] and PalletReady[1] and linea≠2 and PalletEnd[1]≟ False "
      if (LineaHabilitada[1]  and  PalletReady[1]  and  linea != 2  and  PalletEnd[1] ==   False  ):
        $ 415 "oB2V =parpadeo"
        oB2V =parpadeo
        $ 416 "oB2R = False "
        oB2R =  False
      end
      $ 417 "If LineaHabilitada[1] and PalletReady[1] and linea≟2 and PalletEnd[1]≟ False "
      if (LineaHabilitada[1]  and  PalletReady[1]  and  linea == 2  and  PalletEnd[1] ==   False  ):
        $ 418 "oB2V = True "
        oB2V =  True
        $ 419 "oB2R = False "
        oB2R =  False
      end
      $ 420 "Alarmas"
      $ 421 "If AlarmaQM2 or AlarmaVF2 or AlarmaVacio"
      if (AlarmaQM2  or  AlarmaVF2  or  AlarmaVacio):
        $ 422 "Alarma = True "
        Alarma =  True
        $ 423 "StepCode = 98"
        StepCode = 98
      end
      $ 424 "Reset Alarmas"
      $ 425 "If ResetAlarmas"
      if (ResetAlarmas):
        $ 426 "write_output_boolean_register(16,False)"
        write_output_boolean_register(16,False)
        $ 427 "'Reset Alarmas = False'"
        # 'Reset Alarmas = False'
        $ 428 "Alarma=False"
        Alarma=False
        $ 429 "AlarmaVacio = False"
        AlarmaVacio = False
        $ 430 "AlarmaQM1 = False "
        AlarmaQM1 =  False
        $ 431 "AlarmaQM2 = False "
        AlarmaQM2 =  False
        $ 432 "AlarmaVF1 = False "
        AlarmaVF1 =  False
        $ 433 "AlarmaVF2 = False "
        AlarmaVF2 =  False
        $ 434 "temp_alarmas = [0,0,0,0,0,0,0,0,0,0,0,0,0,0,0,0,0,0,0,0,0,0,0,0,0,0,0,0,0,0,0,0,0,0,0,0,0,0,0,0,0,0,0,0,0,0,0,0,0,0]"
        temp_alarmas = [0,0,0,0,0,0,0,0,0,0,0,0,0,0,0,0,0,0,0,0,0,0,0,0,0,0,0,0,0,0,0,0,0,0,0,0,0,0,0,0,0,0,0,0,0,0,0,0,0,0]
      end
      $ 435 "Thread_Avisos"
      $ 436 "Falta colocar palet"
      $ 437 "If  not (iFT1)"
      if (  not  (iFT1)):
        $ 438 "AvisoPaletL1 =  True "
        AvisoPaletL1 =   True
      else:
        $ 439 "Else" "noBreak"
        $ 440 "AvisoPaletL1 =  False "
        AvisoPaletL1 =   False
      end
      $ 441 "If  not (iFT2)"
      if (  not  (iFT2)):
        $ 442 "AvisoPaletL2 =  True "
        AvisoPaletL2 =   True
      else:
        $ 443 "Else" "noBreak"
        $ 444 "AvisoPaletL2 =  False "
        AvisoPaletL2 =   False
      end
      $ 445 "Palet completo"
      $ 446 "If PalletEnd[0]"
      if (PalletEnd[0]):
        $ 447 "AvisoPaletCompletoL1 =  True "
        AvisoPaletCompletoL1 =   True
      else:
        $ 448 "Else" "noBreak"
        $ 449 "AvisoPaletCompletoL1 =  False "
        AvisoPaletCompletoL1 =   False
      end
      $ 450 "If PalletEnd[1]"
      if (PalletEnd[1]):
        $ 451 "AvisoPaletCompletoL2 =  True "
        AvisoPaletCompletoL2 =   True
      else:
        $ 452 "Else" "noBreak"
        $ 453 "AvisoPaletCompletoL2 =  False "
        AvisoPaletCompletoL2 =   False
      end
      $ 454 "Linea Deshabilitada"
      $ 455 "If LineaHabilitada[0]≟ False "
      if (LineaHabilitada[0] ==   False  ):
        $ 456 "AvisoL1Deshab =  True "
        AvisoL1Deshab =   True
      else:
        $ 457 "Else" "noBreak"
        $ 458 "AvisoL1Deshab =  False "
        AvisoL1Deshab =   False
      end
      $ 459 "If LineaHabilitada[1]≟ False "
      if (LineaHabilitada[1] ==   False  ):
        $ 460 "AvisoL2Deshab =  True "
        AvisoL2Deshab =   True
      else:
        $ 461 "Else" "noBreak"
        $ 462 "AvisoL2Deshab =  False "
        AvisoL2Deshab =   False
      end
      $ 463 "SAI sin Servicio"
      $ 464 "If iAVISO_SAI"
      if (iAVISO_SAI):
        $ 465 "StepCode = 90"
        StepCode = 90
        $ 466 "Popup: SAI sin Servicio, el robot se apagara cuando termine el ciclo de dejada"
        popup("SAI sin Servicio, el robot se apagara cuando termine el ciclo de dejada", "Advertencia", True, False, blocking=True)
      end
      $ 467 "If AvisoPaletCompletoL1 or AvisoPaletCompletoL2 or AvisoL1Deshab or AvisoL2Deshab or AvisoPaletL1 or AvisoPaletL2"
      if (AvisoPaletCompletoL1 or AvisoPaletCompletoL2 or AvisoL1Deshab or AvisoL2Deshab or AvisoPaletL1 or AvisoPaletL2):
        $ 468 "Aviso = True"
        Aviso = True
      else:
        $ 469 "Else" "noBreak"
        $ 470 "Aviso =  False "
        Aviso =   False
      end
      $ 471 "sleep(retraso)"
      sleep(retraso)
    end
  end
  threadId_Thread_1 = run Thread_1()
  while (True):
    $ 10 "Robot Program"
    $ 11 "Set Permiso_off=Encender"
    set_configurable_digital_out(5, True)
    $ 12 "If  not (Alarma)"
    if (  not  (Alarma)):
      $ 13 "linea_ant=linea"
      linea_ant=linea
      $ 14 "If ManoConProd≟ False and ManoConCarton≟False"
      if (ManoConProd ==   False  and ManoConCarton == False):
        $ 15 "StepCode = 4"
        StepCode = 4
        $ 16 "Wait LineaPreparada[0] or LineaPreparada[1] or CambioPrograma or CambiosAvanzados"
        while (not(LineaPreparada[0]  or  LineaPreparada[1]  or  CambioPrograma or CambiosAvanzados)):
          sync()
        end
        $ 17 "Loop LineaPreparada[0]≟ False  and LineaPreparada[1]≟ False "
        while (LineaPreparada[0] ==   False    and  LineaPreparada[1] ==   False  ):
          $ 18 "StepCode = 4"
          StepCode = 4
          $ 19 "Wait LineaPreparada[0] or LineaPreparada[1] or CambioPrograma or CambiosAvanzados"
          while (not(LineaPreparada[0]  or  LineaPreparada[1]  or  CambioPrograma or CambiosAvanzados)):
            sync()
          end
          $ 20 "If CambioPrograma or CambiosAvanzados"
          if (CambioPrograma or CambiosAvanzados):
            $ 21 "Call Cambios"
            Cambios()
            $ 22 "Call CargarDatos"
            CargarDatos()
            $ 23 "Script: Calculos_perch.script_bak_bak"
            local j = 0

            yPPerchDejada_min_array = [1,1]
            yPPerchDejada_max_array = [0,0]
            xPPerchDejada_array = [1,1]

            local punto_aux = P_Tipo1[j]
            yPPerchDejada_min_array[0] = punto_aux[1]
            yPPerchDejada_max_array[0] = punto_aux[1]
            xPPerchDejada_array[0] = punto_aux[0]

             while j < Rec_NMovsCapa[Programa_1-1]:
             #while j < 15:
                if punto_aux[1] < yPPerchDejada_min_array[0]:
                    yPPerchDejada_min_array[0] = punto_aux[1]
                end
                if punto_aux[1] > yPPerchDejada_max_array[0]:
                    yPPerchDejada_max_array[0] = punto_aux[1]
                end
                if punto_aux[0] < xPPerchDejada_array[0]:
                   xPPerchDejada_array[0] = punto_aux[0]
                end
                j = j + 1
                punto_aux = P_Tipo1[j]
                sleep(0.01)
            end

            if Rec_CapasTrab[Programa_1-1]:

            	j = 0

            	punto_aux = P_Tipo2[j]
            	yPPerchDejada_min_array[1] = punto_aux[1]
            	yPPerchDejada_max_array[1] = punto_aux[1]
            	xPPerchDejada_array[1] = punto_aux[0]

            	while j < Rec_NMovsCapa[Programa_1-1]:
            #while j < 15:
                		if punto_aux[1] < yPPerchDejada_min_array[1]:
                    			yPPerchDejada_min_array[1] = punto_aux[1]
                		end
                		if punto_aux[1] > yPPerchDejada_max_array[1]:
                    			yPPerchDejada_max_array[1] = punto_aux[1]
                		end
                		if punto_aux[0] < xPPerchDejada_array[1]:
                   			xPPerchDejada_array[1] = punto_aux[0]
                		end
                		j = j + 1
                		punto_aux = P_Tipo2[j]
                		sleep(0.01)
            	end

            end

            if yPPerchDejada_min_array[1]<yPPerchDejada_min_array[0]:
            	global yPPerchDejada_min = yPPerchDejada_min_array[1]
            else:
            	global yPPerchDejada_min = yPPerchDejada_min_array[0]
            end

            if yPPerchDejada_max_array[1]>yPPerchDejada_max_array[0]:
            	global yPPerchDejada_max = yPPerchDejada_max_array[1]
            else:
            	global yPPerchDejada_max = yPPerchDejada_max_array[0]
            end

            if xPPerchDejada_array[1]<xPPerchDejada_array[0]:
            	global xPPerchDejada = xPPerchDejada_array[1]
            else:
            	global xPPerchDejada = xPPerchDejada_array[0]
  global Movs2en2_M1_T1=[False, False, False, False, False, False, False, False, False, False, False, False, False, False, False, False, False, False, False, False, False, False, False, False, False]
  global Movs2en2_M1_T2=[False, False, False, False, False, False, False, False, False, False, False, False, False, False, False, False, False, False, False, False, False, False, False, False, False]
  global ordenM2_T1=[7, 8, 9, 10, 12, 11, 2, 1, 3, 4, 5, 6, 1, 1, 1, 1, 1, 1, 1, 1, 1, 1, 1, 1, 1]
  global ordenM2_T2=[8, 7, 9, 10, 11, 12, 1, 2, 3, 4, 6, 5, 1, 1, 1, 1, 1, 1, 1, 1, 1, 1, 1, 1, 1]
  global Movs2en2_M2_T1=[False, False, False, False, False, False, False, False, False, False, False, False, False, False, False, False, False, False, False, False, False, False, False, False, False]
  global Movs2en2_M2_T2=[False, False, False, False, False, False, False, False, False, False, False, False, False, False, False, False, False, False, False, False, False, False, False, False, False]
  global ordenM3_T1=[6, 7, 1, 2, 3, 4, 5, 1, 1, 1, 1, 1, 1, 1, 1, 1, 1, 1, 1, 1, 1, 1, 1, 1, 1]
  global ordenM3_T2=[3, 4, 5, 6, 7, 1, 2, 1, 1, 1, 1, 1, 1, 1, 1, 1, 1, 1, 1, 1, 1, 1, 1, 1, 1]
  global Movs2en2_M3_T1=[False, False, False, False, False, False, False, False, False, False, False, False, False, False, False, False, False, False, False, False, False, False, False, False, False]
  global Movs2en2_M3_T2=[False, False, False, False, False, False, False, False, False, False, False, False, False, False, False, False, False, False, False, False, False, False, False, False, False]
  global Rec_NMovsCapa=[32, 32, 0, 0, 0, 0, 0, 0, 0, 0]
  global Rec_Cogida2en2=[False, False, False, False, False, False, False, False, False, False]
  global Rec_Carton=[False, False, False, False, False, False, False, False, False, False]
  global Rec_LargoPrd=[280, 280, 0, 0, 0, 0, 0, 0, 0, 0]
  global Rec_AnchoPrd=[97, 97, 0, 0, 0, 0, 0, 0, 0, 0]
  global Rec_AltoPrd=[160, 160, 0, 0, 0, 0, 0, 0, 0, 0]
            end


            if Rec_CapasTrab[Programa_1-1] == True:
            	Rec_TipoCapa = [1, 2, 1, 2, 1, 2, 1, 2, 1, 2, 1, 2, 1, 2, 1, 2, 1, 2, 1, 2, 1, 2, 1, 2, 1, 2, 1, 2, 1, 2]

            else:
            	Rec_TipoCapa = [1,1,1,1,1,1,1,1,1,1,1,1,1,1,1,1,1,1,1,1,1,1,1,1,1,1,1,1,1,1]
            end


            #Dónde poner cartón en función del Programa_1
            #if Programa_1 == 12:
            	#Rec_Carton = #[True,False,False,True,False,False,True,False,False,True,False,False,True,False,False,True,False,False,True,False,False,True,False,False,True,False,False,True,False,False]

            #else:
            	#Rec_Carton = #[False,False,False,False,False,False,False,False,False,False,False,False,False,False,False,False,False,False,False,False,False,False,False,False,False,False,False,False,False,False]
            #end
          end
          $ 24 "sleep(retraso)"
          sleep(retraso)
        end
        $ 25 "If (LineaPreparada[0] and  not LineaPreparada[1]) or ((LineaPreparada[0] and LineaPreparada[1]) and linea_ant≟1)"
        if ((LineaPreparada[0]  and    not  LineaPreparada[1])  or  ((LineaPreparada[0]  and  LineaPreparada[1])  and  linea_ant == 1)):
          $ 26 "linea = 1"
          linea = 1
        else:
          $ 27 "Else" "noBreak"
          $ 28 "linea = 2"
          linea = 2
        end
      end
      $ 29 "Call CargarDatos"
      CargarDatos()
      $ 30 "Call Calculos"
      Calculos()
      $ 31 "Call Movimientos"
      Movimientos()
    end
  end
end
